LIN {X 0,Y 523.999,Z 356.213,A -85,B 0,C 180,E1 -4851.516,E2 -4851.516} C_VEL
LIN {X 0,Y 524.077,Z 356.199,A -85,B 0,C 180,E1 -4854.614,E2 -4854.614} C_VEL
LIN {X 0,Y 524.103,Z 356.198,A -85,B 0,C 180,E1 -4857.695,E2 -4857.695} C_VEL
LIN {X 0,Y 524.118,Z 356.196,A -85,B 0,C 180,E1 -4860.769,E2 -4860.769} C_VEL
LIN {X 0,Y 524.069,Z 356.203,A -85,B 0,C 180,E1 -4863.075,E2 -4863.075} C_VEL
LIN {X 0,Y 524.038,Z 356.203,A -85,B 0,C 180,E1 -4866.159,E2 -4866.159} C_VEL
LIN {X 0,Y 523.997,Z 356.217,A -85,B 0,C 180,E1 -4869.262,E2 -4869.262} C_VEL
LIN {X 0,Y 523.999,Z 356.208,A -85,B 0,C 180,E1 -4871.743,E2 -4871.743} C_VEL
LIN {X 0,Y 523.984,Z 356.219,A -85,B 0,C 180,E1 -4875.053,E2 -4875.053} C_VEL
LIN {X 0,Y 523.957,Z 356.214,A -85,B 0,C 180,E1 -4877.97,E2 -4877.97} C_VEL
LIN {X 0,Y 523.966,Z 356.212,A -85,B 0,C 180,E1 -4880.411,E2 -4880.411} C_VEL
LIN {X 0,Y 523.937,Z 356.224,A -85,B 0,C 180,E1 -4882.893,E2 -4882.893} C_VEL
LIN {X 0,Y 523.979,Z 356.211,A -85,B 0,C 180,E1 -4886.021,E2 -4886.021} C_VEL
LIN {X 0,Y 523.935,Z 356.225,A -85,B 0,C 180,E1 -4888.875,E2 -4888.875} C_VEL
LIN {X 0,Y 523.926,Z 356.22,A -85,B 0,C 180,E1 -4891.544,E2 -4891.544} C_VEL
LIN {X 0,Y 523.941,Z 356.214,A -85,B 0,C 180,E1 -4894.29,E2 -4894.29} C_VEL
LIN {X 0,Y 523.908,Z 356.225,A -85,B 0,C 180,E1 -4897.133,E2 -4897.133} C_VEL
LIN {X 0,Y 523.965,Z 356.214,A -85,B 0,C 180,E1 -4900.135,E2 -4900.135} C_VEL
LIN {X 0,Y 523.924,Z 356.223,A -85,B 0,C 180,E1 -4903.167,E2 -4903.167} C_VEL
LIN {X 0,Y 523.939,Z 356.217,A -85,B 0,C 180,E1 -4905.773,E2 -4905.773} C_VEL
LIN {X 0,Y 523.921,Z 356.223,A -85,B 0,C 180,E1 -4906.927,E2 -4906.927} C_VEL
LIN {X 0,Y 523.254,Z 356.304,A -85,B 0,C 180,E1 -4907.569,E2 -4907.569} C_VEL
LIN {X 0,Y 520.409,Z 356.664,A -85,B 0,C 180,E1 -4908.61,E2 -4908.61} C_VEL
LIN {X 0,Y 518.003,Z 356.963,A -85,B 0,C 180,E1 -4909.449,E2 -4909.449} C_VEL
LIN {X 0,Y 516.967,Z 357.09,A -85,B 0,C 180,E1 -4910.097,E2 -4910.097} C_VEL
LIN {X 0,Y 516.881,Z 357.101,A -85,B 0,C 180,E1 -4910.316,E2 -4910.316} C_VEL
LIN {X 0,Y 516.886,Z 357.102,A -85,B 0,C 180,E1 -4913.343,E2 -4913.343} C_VEL
LIN {X 0,Y 516.918,Z 357.18,A -85,B 0,C 180,E1 -4914.701,E2 -4914.701} C_VEL
LIN {X 0,Y 517.572,Z 361.395,A -85,B 0,C 180,E1 -4915.619,E2 -4915.619} C_VEL
LIN {X 0,Y 517.269,Z 376.326,A -85,B 0,C 180,E1 -4918.704,E2 -4918.704} C_VEL
LIN {X 0,Y 519.142,Z 386.126,A -85,B 0,C 180,E1 -4918.9,E2 -4918.9} C_VEL
LIN {X 0,Y 518.653,Z 482.307,A -85,B 0,C 180,E1 -4920.255,E2 -4920.255} C_VEL
LIN {X 0,Y 518.435,Z 495.531,A -85,B 0,C 180,E1 -4920.598,E2 -4920.598} C_VEL
LIN {X 0,Y 518.202,Z 508.654,A -85,B 0,C 180,E1 -4921.109,E2 -4921.109} C_VEL
LIN {X 0,Y 517.932,Z 520.368,A -85,B 0,C 180,E1 -4921.735,E2 -4921.735} C_VEL
LIN {X 0,Y 517.624,Z 531.628,A -85,B 0,C 180,E1 -4922.508,E2 -4922.508} C_VEL
LIN {X 0,Y 517.32,Z 541.648,A -85,B 0,C 180,E1 -4923.365,E2 -4923.365} C_VEL
LIN {X 0,Y 517.089,Z 549.864,A -85,B 0,C 180,E1 -4924.22,E2 -4924.22} C_VEL
LIN {X 0,Y 516.865,Z 558.043,A -85,B 0,C 180,E1 -4925.245,E2 -4925.245} C_VEL
LIN {X 0,Y 516.666,Z 565.201,A -85,B 0,C 180,E1 -4926.343,E2 -4926.343} C_VEL
LIN {X 0,Y 516.487,Z 572.285,A -85,B 0,C 180,E1 -4927.715,E2 -4927.715} C_VEL
LIN {X 0,Y 516.365,Z 576.909,A -85,B 0,C 180,E1 -4928.859,E2 -4928.859} C_VEL
LIN {X 0,Y 516.33,Z 580.762,A -85,B 0,C 180,E1 -4930.106,E2 -4930.106} C_VEL
LIN {X 0,Y 516.212,Z 582.707,A -85,B 0,C 180,E1 -4930.929,E2 -4930.929} C_VEL
LIN {X 0,Y 516.222,Z 584.92,A -85,B 0,C 180,E1 -4932.366,E2 -4932.366} C_VEL
LIN {X 0,Y 516.168,Z 585.709,A -85,B 0,C 180,E1 -4933.386,E2 -4933.386} C_VEL
LIN {X 0,Y 516.138,Z 585.826,A -85,B 0,C 180,E1 -4934.197,E2 -4934.197} C_VEL
LIN {X 0,Y 516.207,Z 585.427,A -85,B 0,C 180,E1 -4935.162,E2 -4935.162} C_VEL
LIN {X 0,Y 516.202,Z 583.697,A -85,B 0,C 180,E1 -4936.618,E2 -4936.618} C_VEL
LIN {X 0,Y 516.302,Z 581.187,A -85,B 0,C 180,E1 -4937.82,E2 -4937.82} C_VEL
LIN {X 0,Y 516.375,Z 577.665,A -85,B 0,C 180,E1 -4939.016,E2 -4939.016} C_VEL
LIN {X 0,Y 516.454,Z 573.038,A -85,B 0,C 180,E1 -4940.206,E2 -4940.206} C_VEL
LIN {X 0,Y 516.62,Z 566.055,A -85,B 0,C 180,E1 -4941.591,E2 -4941.591} C_VEL
LIN {X 0,Y 516.858,Z 558.51,A -85,B 0,C 180,E1 -4942.775,E2 -4942.775} C_VEL
LIN {X 0,Y 517.094,Z 549.072,A -85,B 0,C 180,E1 -4943.954,E2 -4943.954} C_VEL
LIN {X 0,Y 517.352,Z 539.351,A -85,B 0,C 180,E1 -4944.934,E2 -4944.934} C_VEL
LIN {X 0,Y 517.682,Z 528.486,A -85,B 0,C 180,E1 -4945.815,E2 -4945.815} C_VEL
LIN {X 0,Y 517.98,Z 517.863,A -85,B 0,C 180,E1 -4946.5,E2 -4946.5} C_VEL
LIN {X 0,Y 518.301,Z 505.089,A -85,B 0,C 180,E1 -4947.134,E2 -4947.134} C_VEL
LIN {X 0,Y 518.516,Z 492.947,A -85,B 0,C 180,E1 -4947.572,E2 -4947.572} C_VEL
LIN {X 0,Y 518.672,Z 480.556,A -85,B 0,C 180,E1 -4947.865,E2 -4947.865} C_VEL
LIN {X 0,Y 519.047,Z 385.536,A -85,B 0,C 180,E1 -4949.2,E2 -4949.2} C_VEL
LIN {X 0,Y 517.211,Z 376.145,A -85,B 0,C 180,E1 -4949.392,E2 -4949.392} C_VEL
LIN {X 0,Y 517.596,Z 361.894,A -85,B 0,C 180,E1 -4952.335,E2 -4952.335} C_VEL
LIN {X 0,Y 516.966,Z 357.094,A -85,B 0,C 180,E1 -4953.41,E2 -4953.41} C_VEL
LIN {X 0,Y 516.995,Z 357.083,A -85,B 0,C 180,E1 -4956.243,E2 -4956.243} C_VEL
LIN {X 0,Y 516.955,Z 357.095,A -85,B 0,C 180,E1 -4959.389,E2 -4959.389} C_VEL
LIN {X 0,Y 516.958,Z 357.088,A -85,B 0,C 180,E1 -4961.807,E2 -4961.807} C_VEL
LIN {X 0,Y 516.95,Z 357.092,A -85,B 0,C 180,E1 -4965.146,E2 -4965.146} C_VEL
LIN {X 0,Y 516.929,Z 357.089,A -85,B 0,C 180,E1 -4968.222,E2 -4968.222} C_VEL
LIN {X 0,Y 516.917,Z 357.092,A -85,B 0,C 180,E1 -4970.701,E2 -4970.701} C_VEL
LIN {X 0,Y 516.915,Z 357.091,A -85,B 0,C 180,E1 -4974.071,E2 -4974.071} C_VEL
LIN {X 0,Y 516.928,Z 357.091,A -85,B 0,C 180,E1 -4976.657,E2 -4976.657} C_VEL
LIN {X 0,Y 516.914,Z 357.095,A -85,B 0,C 180,E1 -4979.523,E2 -4979.523} C_VEL
LIN {X 0,Y 516.902,Z 357.093,A -85,B 0,C 180,E1 -4982.543,E2 -4982.543} C_VEL
LIN {X 0,Y 516.884,Z 357.101,A -85,B 0,C 180,E1 -4985.331,E2 -4985.331} C_VEL
LIN {X 0,Y 516.882,Z 357.095,A -85,B 0,C 180,E1 -4987.942,E2 -4987.942} C_VEL
LIN {X 0,Y 516.885,Z 357.098,A -85,B 0,C 180,E1 -4990.74,E2 -4990.74} C_VEL
LIN {X 0,Y 516.883,Z 357.1,A -85,B 0,C 180,E1 -4992.83,E2 -4992.83} C_VEL
LIN {X 0,Y 516.92,Z 357.099,A -85,B 0,C 180,E1 -4995.009,E2 -4995.009} C_VEL
LIN {X 0,Y 516.915,Z 357.092,A -85,B 0,C 180,E1 -4998.397,E2 -4998.397} C_VEL
LIN {X 0,Y 516.88,Z 357.099,A -85,B 0,C 180,E1 -5001.283,E2 -5001.283} C_VEL
LIN {X 0,Y 516.886,Z 357.095,A -85,B 0,C 180,E1 -5004.22,E2 -5004.22} C_VEL
LIN {X 0,Y 516.893,Z 357.1,A -85,B 0,C 180,E1 -5007.052,E2 -5007.052} C_VEL
LIN {X 0,Y 516.887,Z 357.094,A -85,B 0,C 180,E1 -5009.795,E2 -5009.795} C_VEL
LIN {X 0,Y 516.924,Z 357.093,A -85,B 0,C 180,E1 -5012.467,E2 -5012.467} C_VEL
LIN {X 0,Y 516.905,Z 357.097,A -85,B 0,C 180,E1 -5015.071,E2 -5015.071} C_VEL
LIN {X 0,Y 516.879,Z 357.1,A -85,B 0,C 180,E1 -5018.462,E2 -5018.462} C_VEL
LIN {X 0,Y 516.898,Z 357.098,A -85,B 0,C 180,E1 -5020.954,E2 -5020.954} C_VEL
LIN {X 0,Y 516.91,Z 357.092,A -85,B 0,C 180,E1 -5023.41,E2 -5023.41} C_VEL
LIN {X 0,Y 516.887,Z 357.094,A -85,B 0,C 180,E1 -5025.833,E2 -5025.833} C_VEL
LIN {X 0,Y 516.956,Z 357.089,A -85,B 0,C 180,E1 -5028.233,E2 -5028.233} C_VEL
LIN {X 0,Y 516.964,Z 357.085,A -85,B 0,C 180,E1 -5031.399,E2 -5031.399} C_VEL
LIN {X 0,Y 517.035,Z 357.084,A -85,B 0,C 180,E1 -5034.54,E2 -5034.54} C_VEL
LIN {X 0,Y 517.075,Z 357.071,A -85,B 0,C 180,E1 -5037.663,E2 -5037.663} C_VEL
LIN {X 0,Y 517.086,Z 357.074,A -85,B 0,C 180,E1 -5040.779,E2 -5040.779} C_VEL
LIN {X 0,Y 517.008,Z 357.08,A -85,B 0,C 180,E1 -5043.117,E2 -5043.117} C_VEL
LIN {X 0,Y 517.001,Z 357.086,A -85,B 0,C 180,E1 -5046.243,E2 -5046.243} C_VEL
LIN {X 0,Y 516.949,Z 357.086,A -85,B 0,C 180,E1 -5049.389,E2 -5049.389} C_VEL
LIN {X 0,Y 516.947,Z 357.088,A -85,B 0,C 180,E1 -5051.81,E2 -5051.81} C_VEL
LIN {X 0,Y 516.934,Z 357.089,A -85,B 0,C 180,E1 -5055.147,E2 -5055.147} C_VEL
LIN {X 0,Y 516.917,Z 357.098,A -85,B 0,C 180,E1 -5058.222,E2 -5058.222} C_VEL
LIN {X 0,Y 516.904,Z 357.095,A -85,B 0,C 180,E1 -5060.702,E2 -5060.702} C_VEL
LIN {X 0,Y 516.903,Z 357.098,A -85,B 0,C 180,E1 -5064.072,E2 -5064.072} C_VEL
LIN {X 0,Y 516.921,Z 357.093,A -85,B 0,C 180,E1 -5066.658,E2 -5066.658} C_VEL
LIN {X 0,Y 516.917,Z 357.091,A -85,B 0,C 180,E1 -5069.527,E2 -5069.527} C_VEL
LIN {X 0,Y 516.894,Z 357.097,A -85,B 0,C 180,E1 -5072.545,E2 -5072.545} C_VEL
LIN {X 0,Y 516.877,Z 357.096,A -85,B 0,C 180,E1 -5075.333,E2 -5075.333} C_VEL
LIN {X 0,Y 516.876,Z 357.102,A -85,B 0,C 180,E1 -5077.944,E2 -5077.944} C_VEL
LIN {X 0,Y 516.899,Z 357.094,A -85,B 0,C 180,E1 -5080.74,E2 -5080.74} C_VEL
LIN {X 0,Y 516.878,Z 357.102,A -85,B 0,C 180,E1 -5083.904,E2 -5083.904} C_VEL
LIN {X 0,Y 516.878,Z 357.103,A -85,B 0,C 180,E1 -5086.108,E2 -5086.108} C_VEL
LIN {X 0,Y 516.909,Z 357.092,A -85,B 0,C 180,E1 -5089.262,E2 -5089.262} C_VEL
LIN {X 0,Y 516.88,Z 357.102,A -85,B 0,C 180,E1 -5092.057,E2 -5092.057} C_VEL
LIN {X 0,Y 516.894,Z 357.094,A -85,B 0,C 180,E1 -5095.177,E2 -5095.177} C_VEL
LIN {X 0,Y 516.883,Z 357.102,A -85,B 0,C 180,E1 -5097.977,E2 -5097.977} C_VEL
LIN {X 0,Y 516.936,Z 357.091,A -85,B 0,C 180,E1 -5100.697,E2 -5100.697} C_VEL
LIN {X 0,Y 516.943,Z 357.097,A -85,B 0,C 180,E1 -5103.804,E2 -5103.804} C_VEL
LIN {X 0,Y 516.979,Z 357.292,A -85,B 0,C 180,E1 -5104.754,E2 -5104.754} C_VEL
LIN {X 0,Y 518.678,Z 366.12,A -85,B 0,C 180,E1 -5106.228,E2 -5106.228} C_VEL
LIN {X 0,Y 518.204,Z 383.61,A -85,B 0,C 180,E1 -5108.937,E2 -5108.937} C_VEL
LIN {X 0,Y 517.69,Z 403.523,A -85,B 0,C 180,E1 -5111.973,E2 -5111.973} C_VEL
LIN {X 0,Y 517.314,Z 421.232,A -85,B 0,C 180,E1 -5114.631,E2 -5114.631} C_VEL
LIN {X 0,Y 519.105,Z 433.679,A -85,B 0,C 180,E1 -5114.86,E2 -5114.86} C_VEL
LIN {X 0,Y 518.63,Z 529.582,A -85,B 0,C 180,E1 -5116.207,E2 -5116.207} C_VEL
LIN {X 0,Y 518.369,Z 542.929,A -85,B 0,C 180,E1 -5116.55,E2 -5116.55} C_VEL
LIN {X 0,Y 518.05,Z 556.268,A -85,B 0,C 180,E1 -5117.065,E2 -5117.065} C_VEL
LIN {X 0,Y 517.745,Z 568.697,A -85,B 0,C 180,E1 -5117.733,E2 -5117.733} C_VEL
LIN {X 0,Y 517.479,Z 580.404,A -85,B 0,C 180,E1 -5118.544,E2 -5118.544} C_VEL
LIN {X 0,Y 517.163,Z 590.635,A -85,B 0,C 180,E1 -5119.429,E2 -5119.429} C_VEL
LIN {X 0,Y 516.901,Z 599.843,A -85,B 0,C 180,E1 -5120.413,E2 -5120.413} C_VEL
LIN {X 0,Y 516.667,Z 608.817,A -85,B 0,C 180,E1 -5121.592,E2 -5121.592} C_VEL
LIN {X 0,Y 516.509,Z 616.042,A -85,B 0,C 180,E1 -5122.77,E2 -5122.77} C_VEL
LIN {X 0,Y 516.423,Z 622.625,A -85,B 0,C 180,E1 -5124.142,E2 -5124.142} C_VEL
LIN {X 0,Y 516.271,Z 626.976,A -85,B 0,C 180,E1 -5125.315,E2 -5125.315} C_VEL
LIN {X 0,Y 516.37,Z 629.286,A -85,B 0,C 180,E1 -5126.098,E2 -5126.098} C_VEL
LIN {X 0,Y 516.282,Z 631.152,A -85,B 0,C 180,E1 -5126.879,E2 -5126.879} C_VEL
LIN {X 0,Y 516.26,Z 632.552,A -85,B 0,C 180,E1 -5127.659,E2 -5127.659} C_VEL
LIN {X 0,Y 516.16,Z 634.157,A -85,B 0,C 180,E1 -5129.22,E2 -5129.22} C_VEL
LIN {X 0,Y 516.158,Z 634.374,A -85,B 0,C 180,E1 -5130,E2 -5130} C_VEL
LIN {X 0,Y 516.192,Z 633.547,A -85,B 0,C 180,E1 -5131.56,E2 -5131.56} C_VEL
LIN {X 0,Y 516.26,Z 632.55,A -85,B 0,C 180,E1 -5132.341,E2 -5132.341} C_VEL
LIN {X 0,Y 516.282,Z 631.147,A -85,B 0,C 180,E1 -5133.121,E2 -5133.121} C_VEL
LIN {X 0,Y 516.313,Z 628.198,A -85,B 0,C 180,E1 -5134.293,E2 -5134.293} C_VEL
LIN {X 0,Y 516.376,Z 624.207,A -85,B 0,C 180,E1 -5135.467,E2 -5135.467} C_VEL
LIN {X 0,Y 516.474,Z 618.311,A -85,B 0,C 180,E1 -5136.791,E2 -5136.791} C_VEL
LIN {X 0,Y 516.606,Z 611.362,A -85,B 0,C 180,E1 -5138.015,E2 -5138.015} C_VEL
LIN {X 0,Y 516.798,Z 603.043,A -85,B 0,C 180,E1 -5139.194,E2 -5139.194} C_VEL
LIN {X 0,Y 517.056,Z 594.52,A -85,B 0,C 180,E1 -5140.177,E2 -5140.177} C_VEL
LIN {X 0,Y 517.376,Z 583.992,A -85,B 0,C 180,E1 -5141.161,E2 -5141.161} C_VEL
LIN {X 0,Y 517.655,Z 572.776,A -85,B 0,C 180,E1 -5142.004,E2 -5142.004} C_VEL
LIN {X 0,Y 517.988,Z 562.168,A -85,B 0,C 180,E1 -5142.637,E2 -5142.637} C_VEL
LIN {X 0,Y 518.225,Z 550.45,A -85,B 0,C 180,E1 -5143.179,E2 -5143.179} C_VEL
LIN {X 0,Y 518.473,Z 537.871,A -85,B 0,C 180,E1 -5143.597,E2 -5143.597} C_VEL
LIN {X 0,Y 518.683,Z 525.111,A -85,B 0,C 180,E1 -5143.866,E2 -5143.866} C_VEL
LIN {X 0,Y 518.991,Z 432.34,A -85,B 0,C 180,E1 -5145.161,E2 -5145.161} C_VEL
LIN {X 0,Y 517.327,Z 421.045,A -85,B 0,C 180,E1 -5145.377,E2 -5145.377} C_VEL
LIN {X 0,Y 517.765,Z 399.611,A -85,B 0,C 180,E1 -5148.601,E2 -5148.601} C_VEL
LIN {X 0,Y 518.261,Z 380.763,A -85,B 0,C 180,E1 -5151.477,E2 -5151.477} C_VEL
LIN {X 0,Y 518.63,Z 365.975,A -85,B 0,C 180,E1 -5153.774,E2 -5153.774} C_VEL
LIN {X 0,Y 516.971,Z 357.09,A -85,B 0,C 180,E1 -5155.274,E2 -5155.274} C_VEL
LIN {X 0,Y 516.925,Z 357.098,A -85,B 0,C 180,E1 -5158.414,E2 -5158.414} C_VEL
LIN {X 0,Y 516.892,Z 357.095,A -85,B 0,C 180,E1 -5161.109,E2 -5161.109} C_VEL
LIN {X 0,Y 516.912,Z 357.098,A -85,B 0,C 180,E1 -5163.966,E2 -5163.966} C_VEL
LIN {X 0,Y 516.881,Z 357.098,A -85,B 0,C 180,E1 -5166.745,E2 -5166.745} C_VEL
LIN {X 0,Y 516.909,Z 357.096,A -85,B 0,C 180,E1 -5169.718,E2 -5169.718} C_VEL
LIN {X 0,Y 516.882,Z 357.095,A -85,B 0,C 180,E1 -5172.757,E2 -5172.757} C_VEL
LIN {X 0,Y 516.918,Z 357.091,A -85,B 0,C 180,E1 -5175.009,E2 -5175.009} C_VEL
LIN {X 0,Y 516.918,Z 357.093,A -85,B 0,C 180,E1 -5178.397,E2 -5178.397} C_VEL
LIN {X 0,Y 516.901,Z 357.094,A -85,B 0,C 180,E1 -5181.286,E2 -5181.286} C_VEL
LIN {X 0,Y 516.884,Z 357.098,A -85,B 0,C 180,E1 -5184.221,E2 -5184.221} C_VEL
LIN {X 0,Y 516.891,Z 357.093,A -85,B 0,C 180,E1 -5187.053,E2 -5187.053} C_VEL
LIN {X 0,Y 516.895,Z 357.099,A -85,B 0,C 180,E1 -5189.796,E2 -5189.796} C_VEL
LIN {X 0,Y 516.922,Z 357.09,A -85,B 0,C 180,E1 -5192.467,E2 -5192.467} C_VEL
LIN {X 0,Y 516.903,Z 357.093,A -85,B 0,C 180,E1 -5195.072,E2 -5195.072} C_VEL
LIN {X 0,Y 516.878,Z 357.093,A -85,B 0,C 180,E1 -5198.462,E2 -5198.462} C_VEL
LIN {X 0,Y 516.896,Z 357.095,A -85,B 0,C 180,E1 -5200.955,E2 -5200.955} C_VEL
LIN {X 0,Y 516.909,Z 357.095,A -85,B 0,C 180,E1 -5203.41,E2 -5203.41} C_VEL
LIN {X 0,Y 516.897,Z 357.097,A -85,B 0,C 180,E1 -5205.834,E2 -5205.834} C_VEL
LIN {X 0,Y 516.948,Z 357.088,A -85,B 0,C 180,E1 -5209.028,E2 -5209.028} C_VEL
LIN {X 0,Y 516.969,Z 357.081,A -85,B 0,C 180,E1 -5212.187,E2 -5212.187} C_VEL
LIN {X 0,Y 517.024,Z 357.077,A -85,B 0,C 180,E1 -5214.54,E2 -5214.54} C_VEL
LIN {X 0,Y 517.076,Z 357.074,A -85,B 0,C 180,E1 -5217.663,E2 -5217.663} C_VEL
LIN {X 0,Y 517.088,Z 357.072,A -85,B 0,C 180,E1 -5220.779,E2 -5220.779} C_VEL
LIN {X 0,Y 517.01,Z 357.082,A -85,B 0,C 180,E1 -5223.117,E2 -5223.117} C_VEL
LIN {X 0,Y 517.002,Z 357.079,A -85,B 0,C 180,E1 -5226.243,E2 -5226.243} C_VEL
LIN {X 0,Y 516.951,Z 357.093,A -85,B 0,C 180,E1 -5229.39,E2 -5229.39} C_VEL
LIN {X 0,Y 516.948,Z 357.085,A -85,B 0,C 180,E1 -5231.811,E2 -5231.811} C_VEL
LIN {X 0,Y 516.935,Z 357.095,A -85,B 0,C 180,E1 -5235.147,E2 -5235.147} C_VEL
LIN {X 0,Y 516.919,Z 357.091,A -85,B 0,C 180,E1 -5238.223,E2 -5238.223} C_VEL
LIN {X 0,Y 516.908,Z 357.094,A -85,B 0,C 180,E1 -5240.702,E2 -5240.702} C_VEL
LIN {X 0,Y 516.885,Z 357.099,A -85,B 0,C 180,E1 -5243.223,E2 -5243.223} C_VEL
LIN {X 0,Y 516.938,Z 357.089,A -85,B 0,C 180,E1 -5246.198,E2 -5246.198} C_VEL
LIN {X 0,Y 516.917,Z 357.094,A -85,B 0,C 180,E1 -5249.305,E2 -5249.305} C_VEL
LIN {X 0,Y 516.896,Z 357.098,A -85,B 0,C 180,E1 -5252.545,E2 -5252.545} C_VEL
LIN {X 0,Y 516.879,Z 357.098,A -85,B 0,C 180,E1 -5255.333,E2 -5255.333} C_VEL
LIN {X 0,Y 516.878,Z 357.096,A -85,B 0,C 180,E1 -5257.944,E2 -5257.944} C_VEL
LIN {X 0,Y 516.901,Z 357.101,A -85,B 0,C 180,E1 -5260.741,E2 -5260.741} C_VEL
LIN {X 0,Y 516.881,Z 357.097,A -85,B 0,C 180,E1 -5263.904,E2 -5263.904} C_VEL
LIN {X 0,Y 516.881,Z 357.098,A -85,B 0,C 180,E1 -5266.108,E2 -5266.108} C_VEL
LIN {X 0,Y 516.916,Z 357.096,A -85,B 0,C 180,E1 -5268.399,E2 -5268.399} C_VEL
LIN {X 0,Y 516.881,Z 357.101,A -85,B 0,C 180,E1 -5270.316,E2 -5270.316} C_VEL
LIN {X 0,Y 516.212,Z 357.187,A -85,B 0,C 180,E1 -5270.967,E2 -5270.967} C_VEL
LIN {X 0,Y 513.363,Z 357.541,A -85,B 0,C 180,E1 -5272.022,E2 -5272.022} C_VEL
LIN {X 0,Y 510.955,Z 357.844,A -85,B 0,C 180,E1 -5272.873,E2 -5272.873} C_VEL
LIN {X 0,Y 509.92,Z 357.97,A -85,B 0,C 180,E1 -5273.529,E2 -5273.529} C_VEL
LIN {X 0,Y 509.834,Z 357.98,A -85,B 0,C 180,E1 -5273.752,E2 -5273.752} C_VEL
LIN {X 0,Y 509.867,Z 358.085,A -85,B 0,C 180,E1 -5274.556,E2 -5274.556} C_VEL
LIN {X 0,Y 510.609,Z 363.173,A -85,B 0,C 180,E1 -5275.674,E2 -5275.674} C_VEL
LIN {X 0,Y 510.286,Z 376.497,A -85,B 0,C 180,E1 -5278.466,E2 -5278.466} C_VEL
LIN {X 0,Y 512.262,Z 386.394,A -85,B 0,C 180,E1 -5278.691,E2 -5278.691} C_VEL
LIN {X 0,Y 511.757,Z 483.293,A -85,B 0,C 180,E1 -5280.081,E2 -5280.081} C_VEL
LIN {X 0,Y 511.515,Z 497.109,A -85,B 0,C 180,E1 -5280.455,E2 -5280.455} C_VEL
LIN {X 0,Y 511.291,Z 509.634,A -85,B 0,C 180,E1 -5280.963,E2 -5280.963} C_VEL
LIN {X 0,Y 510.996,Z 521.095,A -85,B 0,C 180,E1 -5281.591,E2 -5281.591} C_VEL
LIN {X 0,Y 510.637,Z 533.044,A -85,B 0,C 180,E1 -5282.434,E2 -5282.434} C_VEL
LIN {X 0,Y 510.326,Z 542.927,A -85,B 0,C 180,E1 -5283.308,E2 -5283.308} C_VEL
LIN {X 0,Y 510.034,Z 551.834,A -85,B 0,C 180,E1 -5284.276,E2 -5284.276} C_VEL
LIN {X 0,Y 509.738,Z 560.967,A -85,B 0,C 180,E1 -5285.503,E2 -5285.503} C_VEL
LIN {X 0,Y 509.568,Z 567.782,A -85,B 0,C 180,E1 -5286.64,E2 -5286.64} C_VEL
LIN {X 0,Y 509.413,Z 573.613,A -85,B 0,C 180,E1 -5287.848,E2 -5287.848} C_VEL
LIN {X 0,Y 509.29,Z 577.911,A -85,B 0,C 180,E1 -5288.975,E2 -5288.975} C_VEL
LIN {X 0,Y 509.233,Z 581.59,A -85,B 0,C 180,E1 -5290.238,E2 -5290.238} C_VEL
LIN {X 0,Y 509.123,Z 584.135,A -85,B 0,C 180,E1 -5291.489,E2 -5291.489} C_VEL
LIN {X 0,Y 509.157,Z 585.233,A -85,B 0,C 180,E1 -5292.322,E2 -5292.322} C_VEL
LIN {X 0,Y 509.088,Z 585.908,A -85,B 0,C 180,E1 -5293.148,E2 -5293.148} C_VEL
LIN {X 0,Y 509.047,Z 586.175,A -85,B 0,C 180,E1 -5293.971,E2 -5293.971} C_VEL
LIN {X 0,Y 509.122,Z 585.816,A -85,B 0,C 180,E1 -5295.083,E2 -5295.083} C_VEL
LIN {X 0,Y 509.107,Z 584.373,A -85,B 0,C 180,E1 -5296.428,E2 -5296.428} C_VEL
LIN {X 0,Y 509.177,Z 582.943,A -85,B 0,C 180,E1 -5297.242,E2 -5297.242} C_VEL
LIN {X 0,Y 509.273,Z 579.919,A -85,B 0,C 180,E1 -5298.468,E2 -5298.468} C_VEL
LIN {X 0,Y 509.331,Z 575.914,A -85,B 0,C 180,E1 -5299.667,E2 -5299.667} C_VEL
LIN {X 0,Y 509.505,Z 569.695,A -85,B 0,C 180,E1 -5301.073,E2 -5301.073} C_VEL
LIN {X 0,Y 509.713,Z 562.938,A -85,B 0,C 180,E1 -5302.274,E2 -5302.274} C_VEL
LIN {X 0,Y 509.932,Z 554.842,A -85,B 0,C 180,E1 -5303.437,E2 -5303.437} C_VEL
LIN {X 0,Y 510.185,Z 545.962,A -85,B 0,C 180,E1 -5304.467,E2 -5304.467} C_VEL
LIN {X 0,Y 510.534,Z 535.379,A -85,B 0,C 180,E1 -5305.46,E2 -5305.46} C_VEL
LIN {X 0,Y 510.849,Z 524.879,A -85,B 0,C 180,E1 -5306.253,E2 -5306.253} C_VEL
LIN {X 0,Y 511.256,Z 513.128,A -85,B 0,C 180,E1 -5306.947,E2 -5306.947} C_VEL
LIN {X 0,Y 511.452,Z 501.053,A -85,B 0,C 180,E1 -5307.49,E2 -5307.49} C_VEL
LIN {X 0,Y 511.682,Z 487.742,A -85,B 0,C 180,E1 -5307.909,E2 -5307.909} C_VEL
LIN {X 0,Y 511.847,Z 472.57,A -85,B 0,C 180,E1 -5308.18,E2 -5308.18} C_VEL
LIN {X 0,Y 512.249,Z 386.404,A -85,B 0,C 180,E1 -5309.398,E2 -5309.398} C_VEL
LIN {X 0,Y 510.241,Z 376.477,A -85,B 0,C 180,E1 -5309.605,E2 -5309.605} C_VEL
LIN {X 0,Y 510.612,Z 363.229,A -85,B 0,C 180,E1 -5312.366,E2 -5312.366} C_VEL
LIN {X 0,Y 510.232,Z 359.582,A -85,B 0,C 180,E1 -5313.158,E2 -5313.158} C_VEL
LIN {X 0,Y 509.917,Z 357.972,A -85,B 0,C 180,E1 -5313.556,E2 -5313.556} C_VEL
LIN {X 0,Y 509.943,Z 357.962,A -85,B 0,C 180,E1 -5316.33,E2 -5316.33} C_VEL
LIN {X 0,Y 509.913,Z 357.966,A -85,B 0,C 180,E1 -5318.72,E2 -5318.72} C_VEL
LIN {X 0,Y 509.91,Z 357.965,A -85,B 0,C 180,E1 -5321.931,E2 -5321.931} C_VEL
LIN {X 0,Y 509.899,Z 357.972,A -85,B 0,C 180,E1 -5325.241,E2 -5325.241} C_VEL
LIN {X 0,Y 509.887,Z 357.967,A -85,B 0,C 180,E1 -5327.998,E2 -5327.998} C_VEL
LIN {X 0,Y 509.854,Z 357.975,A -85,B 0,C 180,E1 -5331.001,E2 -5331.001} C_VEL
LIN {X 0,Y 509.841,Z 357.976,A -85,B 0,C 180,E1 -5333.562,E2 -5333.562} C_VEL
LIN {X 0,Y 509.914,Z 357.963,A -85,B 0,C 180,E1 -5336.378,E2 -5336.378} C_VEL
LIN {X 0,Y 509.879,Z 357.971,A -85,B 0,C 180,E1 -5338.843,E2 -5338.843} C_VEL
LIN {X 0,Y 509.827,Z 357.977,A -85,B 0,C 180,E1 -5341.589,E2 -5341.589} C_VEL
LIN {X 0,Y 509.855,Z 357.971,A -85,B 0,C 180,E1 -5344.412,E2 -5344.412} C_VEL
LIN {X 0,Y 509.82,Z 357.98,A -85,B 0,C 180,E1 -5347.34,E2 -5347.34} C_VEL
LIN {X 0,Y 509.838,Z 357.973,A -85,B 0,C 180,E1 -5350.381,E2 -5350.381} C_VEL
LIN {X 0,Y 509.823,Z 357.983,A -85,B 0,C 180,E1 -5353.061,E2 -5353.061} C_VEL
LIN {X 0,Y 509.828,Z 357.974,A -85,B 0,C 180,E1 -5355.791,E2 -5355.791} C_VEL
LIN {X 0,Y 509.856,Z 357.973,A -85,B 0,C 180,E1 -5358.574,E2 -5358.574} C_VEL
LIN {X 0,Y 509.848,Z 357.971,A -85,B 0,C 180,E1 -5361.785,E2 -5361.785} C_VEL
LIN {X 0,Y 509.841,Z 357.976,A -85,B 0,C 180,E1 -5364.622,E2 -5364.622} C_VEL
LIN {X 0,Y 509.86,Z 357.971,A -85,B 0,C 180,E1 -5367.48,E2 -5367.48} C_VEL
LIN {X 0,Y 509.852,Z 357.972,A -85,B 0,C 180,E1 -5370.273,E2 -5370.273} C_VEL
LIN {X 0,Y 509.881,Z 357.974,A -85,B 0,C 180,E1 -5372.944,E2 -5372.944} C_VEL
LIN {X 0,Y 509.863,Z 357.969,A -85,B 0,C 180,E1 -5375.573,E2 -5375.573} C_VEL
LIN {X 0,Y 509.815,Z 357.976,A -85,B 0,C 180,E1 -5378.148,E2 -5378.148} C_VEL
LIN {X 0,Y 509.858,Z 357.978,A -85,B 0,C 180,E1 -5380.681,E2 -5380.681} C_VEL
LIN {X 0,Y 509.879,Z 357.97,A -85,B 0,C 180,E1 -5383.174,E2 -5383.174} C_VEL
LIN {X 0,Y 509.856,Z 357.97,A -85,B 0,C 180,E1 -5385.634,E2 -5385.634} C_VEL
LIN {X 0,Y 509.909,Z 357.969,A -85,B 0,C 180,E1 -5388.874,E2 -5388.874} C_VEL
LIN {X 0,Y 509.943,Z 357.961,A -85,B 0,C 180,E1 -5392.078,E2 -5392.078} C_VEL
LIN {X 0,Y 509.985,Z 357.961,A -85,B 0,C 180,E1 -5394.464,E2 -5394.464} C_VEL
LIN {X 0,Y 510.046,Z 357.946,A -85,B 0,C 180,E1 -5397.631,E2 -5397.631} C_VEL
LIN {X 0,Y 510.056,Z 357.95,A -85,B 0,C 180,E1 -5400.789,E2 -5400.789} C_VEL
LIN {X 0,Y 509.95,Z 357.959,A -85,B 0,C 180,E1 -5403.16,E2 -5403.16} C_VEL
LIN {X 0,Y 509.969,Z 357.963,A -85,B 0,C 180,E1 -5406.33,E2 -5406.33} C_VEL
LIN {X 0,Y 509.909,Z 357.968,A -85,B 0,C 180,E1 -5408.72,E2 -5408.72} C_VEL
LIN {X 0,Y 509.895,Z 357.968,A -85,B 0,C 180,E1 -5411.932,E2 -5411.932} C_VEL
LIN {X 0,Y 509.884,Z 357.967,A -85,B 0,C 180,E1 -5415.242,E2 -5415.242} C_VEL
LIN {X 0,Y 509.879,Z 357.971,A -85,B 0,C 180,E1 -5418.001,E2 -5418.001} C_VEL
LIN {X 0,Y 509.842,Z 357.972,A -85,B 0,C 180,E1 -5421.002,E2 -5421.002} C_VEL
LIN {X 0,Y 509.828,Z 357.974,A -85,B 0,C 180,E1 -5423.563,E2 -5423.563} C_VEL
LIN {X 0,Y 509.905,Z 357.971,A -85,B 0,C 180,E1 -5426.38,E2 -5426.38} C_VEL
LIN {X 0,Y 509.878,Z 357.968,A -85,B 0,C 180,E1 -5428.844,E2 -5428.844} C_VEL
LIN {X 0,Y 509.819,Z 357.976,A -85,B 0,C 180,E1 -5431.59,E2 -5431.59} C_VEL
LIN {X 0,Y 509.848,Z 357.976,A -85,B 0,C 180,E1 -5434.414,E2 -5434.414} C_VEL
LIN {X 0,Y 509.813,Z 357.976,A -85,B 0,C 180,E1 -5437.341,E2 -5437.341} C_VEL
LIN {X 0,Y 509.856,Z 357.974,A -85,B 0,C 180,E1 -5440.381,E2 -5440.381} C_VEL
LIN {X 0,Y 509.835,Z 357.973,A -85,B 0,C 180,E1 -5443.065,E2 -5443.065} C_VEL
LIN {X 0,Y 509.826,Z 357.979,A -85,B 0,C 180,E1 -5445.793,E2 -5445.793} C_VEL
LIN {X 0,Y 509.863,Z 357.971,A -85,B 0,C 180,E1 -5448.576,E2 -5448.576} C_VEL
LIN {X 0,Y 509.854,Z 357.977,A -85,B 0,C 180,E1 -5451.786,E2 -5451.786} C_VEL
LIN {X 0,Y 509.845,Z 357.972,A -85,B 0,C 180,E1 -5454.624,E2 -5454.624} C_VEL
LIN {X 0,Y 509.865,Z 357.972,A -85,B 0,C 180,E1 -5457.482,E2 -5457.482} C_VEL
LIN {X 0,Y 509.881,Z 357.973,A -85,B 0,C 180,E1 -5460.27,E2 -5460.27} C_VEL
LIN {X 0,Y 509.886,Z 357.972,A -85,B 0,C 180,E1 -5462.945,E2 -5462.945} C_VEL
LIN {X 0,Y 509.936,Z 357.997,A -85,B 0,C 180,E1 -5464.544,E2 -5464.544} C_VEL
LIN {X 0,Y 511.783,Z 368.525,A -85,B 0,C 180,E1 -5466.318,E2 -5466.318} C_VEL
LIN {X 0,Y 511.138,Z 387.871,A -85,B 0,C 180,E1 -5469.347,E2 -5469.347} C_VEL
LIN {X 0,Y 510.575,Z 408.838,A -85,B 0,C 180,E1 -5472.58,E2 -5472.58} C_VEL
LIN {X 0,Y 510.318,Z 420.982,A -85,B 0,C 180,E1 -5474.417,E2 -5474.417} C_VEL
LIN {X 0,Y 512.252,Z 435.53,A -85,B 0,C 180,E1 -5474.683,E2 -5474.683} C_VEL
LIN {X 0,Y 511.735,Z 529.208,A -85,B 0,C 180,E1 -5476.018,E2 -5476.018} C_VEL
LIN {X 0,Y 511.476,Z 542.571,A -85,B 0,C 180,E1 -5476.365,E2 -5476.365} C_VEL
LIN {X 0,Y 511.14,Z 555.919,A -85,B 0,C 180,E1 -5476.887,E2 -5476.887} C_VEL
LIN {X 0,Y 510.824,Z 567.663,A -85,B 0,C 180,E1 -5477.52,E2 -5477.52} C_VEL
LIN {X 0,Y 510.515,Z 578.763,A -85,B 0,C 180,E1 -5478.285,E2 -5478.285} C_VEL
LIN {X 0,Y 510.199,Z 589.245,A -85,B 0,C 180,E1 -5479.183,E2 -5479.183} C_VEL
LIN {X 0,Y 509.903,Z 597.816,A -85,B 0,C 180,E1 -5480.079,E2 -5480.079} C_VEL
LIN {X 0,Y 509.682,Z 605.729,A -85,B 0,C 180,E1 -5481.076,E2 -5481.076} C_VEL
LIN {X 0,Y 509.476,Z 613.459,A -85,B 0,C 180,E1 -5482.271,E2 -5482.271} C_VEL
LIN {X 0,Y 509.317,Z 619.72,A -85,B 0,C 180,E1 -5483.474,E2 -5483.474} C_VEL
LIN {X 0,Y 509.243,Z 625.327,A -85,B 0,C 180,E1 -5484.853,E2 -5484.853} C_VEL
LIN {X 0,Y 509.275,Z 628.953,A -85,B 0,C 180,E1 -5486.044,E2 -5486.044} C_VEL
LIN {X 0,Y 509.201,Z 630.82,A -85,B 0,C 180,E1 -5486.835,E2 -5486.835} C_VEL
LIN {X 0,Y 509.189,Z 632.221,A -85,B 0,C 180,E1 -5487.627,E2 -5487.627} C_VEL
LIN {X 0,Y 509.073,Z 633.825,A -85,B 0,C 180,E1 -5489.209,E2 -5489.209} C_VEL
LIN {X 0,Y 509.069,Z 634.041,A -85,B 0,C 180,E1 -5490,E2 -5490} C_VEL
LIN {X 0,Y 509.112,Z 633.213,A -85,B 0,C 180,E1 -5491.582,E2 -5491.582} C_VEL
LIN {X 0,Y 509.189,Z 632.215,A -85,B 0,C 180,E1 -5492.373,E2 -5492.373} C_VEL
LIN {X 0,Y 509.201,Z 630.811,A -85,B 0,C 180,E1 -5493.165,E2 -5493.165} C_VEL
LIN {X 0,Y 509.206,Z 627.859,A -85,B 0,C 180,E1 -5494.353,E2 -5494.353} C_VEL
LIN {X 0,Y 509.294,Z 623.866,A -85,B 0,C 180,E1 -5495.543,E2 -5495.543} C_VEL
LIN {X 0,Y 509.407,Z 617.828,A -85,B 0,C 180,E1 -5496.914,E2 -5496.914} C_VEL
LIN {X 0,Y 509.551,Z 611.016,A -85,B 0,C 180,E1 -5498.127,E2 -5498.127} C_VEL
LIN {X 0,Y 509.753,Z 602.694,A -85,B 0,C 180,E1 -5499.323,E2 -5499.323} C_VEL
LIN {X 0,Y 510.025,Z 594.168,A -85,B 0,C 180,E1 -5500.319,E2 -5500.319} C_VEL
LIN {X 0,Y 510.387,Z 583.637,A -85,B 0,C 180,E1 -5501.316,E2 -5501.316} C_VEL
LIN {X 0,Y 510.665,Z 572.417,A -85,B 0,C 180,E1 -5502.171,E2 -5502.171} C_VEL
LIN {X 0,Y 511.039,Z 561.805,A -85,B 0,C 180,E1 -5502.812,E2 -5502.812} C_VEL
LIN {X 0,Y 511.297,Z 550.078,A -85,B 0,C 180,E1 -5503.361,E2 -5503.361} C_VEL
LIN {X 0,Y 511.579,Z 536.572,A -85,B 0,C 180,E1 -5503.809,E2 -5503.809} C_VEL
LIN {X 0,Y 511.79,Z 523.149,A -85,B 0,C 180,E1 -5504.082,E2 -5504.082} C_VEL
LIN {X 0,Y 512.112,Z 432.847,A -85,B 0,C 180,E1 -5505.358,E2 -5505.358} C_VEL
LIN {X 0,Y 510.288,Z 420.625,A -85,B 0,C 180,E1 -5505.605,E2 -5505.605} C_VEL
LIN {X 0,Y 510.762,Z 400.629,A -85,B 0,C 180,E1 -5508.657,E2 -5508.657} C_VEL
LIN {X 0,Y 511.307,Z 381.828,A -85,B 0,C 180,E1 -5511.572,E2 -5511.572} C_VEL
LIN {X 0,Y 511.743,Z 368.402,A -85,B 0,C 180,E1 -5513.684,E2 -5513.684} C_VEL
LIN {X 0,Y 510.122,Z 358.973,A -85,B 0,C 180,E1 -5515.282,E2 -5515.282} C_VEL
LIN {X 0,Y 509.936,Z 357.968,A -85,B 0,C 180,E1 -5515.456,E2 -5515.456} C_VEL
LIN {X 0,Y 509.886,Z 357.971,A -85,B 0,C 180,E1 -5518.843,E2 -5518.843} C_VEL
LIN {X 0,Y 509.826,Z 357.977,A -85,B 0,C 180,E1 -5521.589,E2 -5521.589} C_VEL
LIN {X 0,Y 509.852,Z 357.976,A -85,B 0,C 180,E1 -5524.412,E2 -5524.412} C_VEL
LIN {X 0,Y 509.817,Z 357.978,A -85,B 0,C 180,E1 -5527.34,E2 -5527.34} C_VEL
LIN {X 0,Y 509.874,Z 357.972,A -85,B 0,C 180,E1 -5530.378,E2 -5530.378} C_VEL
LIN {X 0,Y 509.82,Z 357.974,A -85,B 0,C 180,E1 -5533.062,E2 -5533.062} C_VEL
LIN {X 0,Y 509.826,Z 357.981,A -85,B 0,C 180,E1 -5535.792,E2 -5535.792} C_VEL
LIN {X 0,Y 509.86,Z 357.971,A -85,B 0,C 180,E1 -5538.575,E2 -5538.575} C_VEL
LIN {X 0,Y 509.853,Z 357.977,A -85,B 0,C 180,E1 -5541.662,E2 -5541.662} C_VEL
LIN {X 0,Y 509.84,Z 357.973,A -85,B 0,C 180,E1 -5544.623,E2 -5544.623} C_VEL
LIN {X 0,Y 509.859,Z 357.973,A -85,B 0,C 180,E1 -5547.481,E2 -5547.481} C_VEL
LIN {X 0,Y 509.874,Z 357.969,A -85,B 0,C 180,E1 -5550.268,E2 -5550.268} C_VEL
LIN {X 0,Y 509.879,Z 357.968,A -85,B 0,C 180,E1 -5552.944,E2 -5552.944} C_VEL
LIN {X 0,Y 509.862,Z 357.976,A -85,B 0,C 180,E1 -5555.574,E2 -5555.574} C_VEL
LIN {X 0,Y 509.814,Z 357.975,A -85,B 0,C 180,E1 -5558.148,E2 -5558.148} C_VEL
LIN {X 0,Y 509.856,Z 357.971,A -85,B 0,C 180,E1 -5560.681,E2 -5560.681} C_VEL
LIN {X 0,Y 509.879,Z 357.968,A -85,B 0,C 180,E1 -5563.175,E2 -5563.175} C_VEL
LIN {X 0,Y 509.864,Z 357.976,A -85,B 0,C 180,E1 -5565.634,E2 -5565.634} C_VEL
LIN {X 0,Y 509.908,Z 357.964,A -85,B 0,C 180,E1 -5568.875,E2 -5568.875} C_VEL
LIN {X 0,Y 509.943,Z 357.957,A -85,B 0,C 180,E1 -5572.078,E2 -5572.078} C_VEL
LIN {X 0,Y 509.975,Z 357.955,A -85,B 0,C 180,E1 -5574.464,E2 -5574.464} C_VEL
LIN {X 0,Y 510.047,Z 357.95,A -85,B 0,C 180,E1 -5577.631,E2 -5577.631} C_VEL
LIN {X 0,Y 510.058,Z 357.948,A -85,B 0,C 180,E1 -5580.79,E2 -5580.79} C_VEL
LIN {X 0,Y 509.952,Z 357.962,A -85,B 0,C 180,E1 -5583.16,E2 -5583.16} C_VEL
LIN {X 0,Y 509.97,Z 357.955,A -85,B 0,C 180,E1 -5586.33,E2 -5586.33} C_VEL
LIN {X 0,Y 509.911,Z 357.964,A -85,B 0,C 180,E1 -5588.721,E2 -5588.721} C_VEL
LIN {X 0,Y 509.896,Z 357.963,A -85,B 0,C 180,E1 -5591.932,E2 -5591.932} C_VEL
LIN {X 0,Y 509.885,Z 357.972,A -85,B 0,C 180,E1 -5595.242,E2 -5595.242} C_VEL
LIN {X 0,Y 509.881,Z 357.968,A -85,B 0,C 180,E1 -5598.002,E2 -5598.002} C_VEL
LIN {X 0,Y 509.85,Z 357.977,A -85,B 0,C 180,E1 -5601.002,E2 -5601.002} C_VEL
LIN {X 0,Y 509.843,Z 357.972,A -85,B 0,C 180,E1 -5603.563,E2 -5603.563} C_VEL
LIN {X 0,Y 509.907,Z 357.966,A -85,B 0,C 180,E1 -5606.38,E2 -5606.38} C_VEL
LIN {X 0,Y 509.872,Z 357.976,A -85,B 0,C 180,E1 -5608.845,E2 -5608.845} C_VEL
LIN {X 0,Y 509.82,Z 357.977,A -85,B 0,C 180,E1 -5611.591,E2 -5611.591} C_VEL
LIN {X 0,Y 509.85,Z 357.97,A -85,B 0,C 180,E1 -5614.414,E2 -5614.414} C_VEL
LIN {X 0,Y 509.815,Z 357.978,A -85,B 0,C 180,E1 -5617.341,E2 -5617.341} C_VEL
LIN {X 0,Y 509.857,Z 357.974,A -85,B 0,C 180,E1 -5620.381,E2 -5620.381} C_VEL
LIN {X 0,Y 509.838,Z 357.979,A -85,B 0,C 180,E1 -5623.065,E2 -5623.065} C_VEL
LIN {X 0,Y 509.829,Z 357.975,A -85,B 0,C 180,E1 -5625.793,E2 -5625.793} C_VEL
LIN {X 0,Y 509.858,Z 357.978,A -85,B 0,C 180,E1 -5628.576,E2 -5628.576} C_VEL
LIN {X 0,Y 509.852,Z 357.976,A -85,B 0,C 180,E1 -5631.787,E2 -5631.787} C_VEL
LIN {X 0,Y 509.834,Z 357.98,A -85,B 0,C 180,E1 -5633.752,E2 -5633.752} C_VEL
LIN {X 0,Y 509.549,Z 358.387,A -85,B 0,C 180,E1 -5634.189,E2 -5634.189} C_VEL
LIN {X 0,Y 508.378,Z 360.147,A -85,B 0,C 180,E1 -5634.812,E2 -5634.812} C_VEL
LIN {X 0,Y 506.757,Z 362.716,A -85,B 0,C 180,E1 -5635.396,E2 -5635.396} C_VEL
LIN {X 0,Y 503.827,Z 368.763,A -85,B 0,C 180,E1 -5636.553,E2 -5636.553} C_VEL
LIN {X 0,Y 503.462,Z 370.709,A -85,B 0,C 180,E1 -5636.952,E2 -5636.952} C_VEL
LIN {X 0,Y 503.328,Z 376.94,A -85,B 0,C 180,E1 -5638.266,E2 -5638.266} C_VEL
LIN {X 0,Y 505.473,Z 388.512,A -85,B 0,C 180,E1 -5638.505,E2 -5638.505} C_VEL
LIN {X 0,Y 504.897,Z 483.205,A -85,B 0,C 180,E1 -5639.879,E2 -5639.879} C_VEL
LIN {X 0,Y 504.66,Z 496.285,A -85,B 0,C 180,E1 -5640.228,E2 -5640.228} C_VEL
LIN {X 0,Y 504.395,Z 509.441,A -85,B 0,C 180,E1 -5640.756,E2 -5640.756} C_VEL
LIN {X 0,Y 504.052,Z 521.965,A -85,B 0,C 180,E1 -5641.452,E2 -5641.452} C_VEL
LIN {X 0,Y 503.714,Z 533.068,A -85,B 0,C 180,E1 -5642.248,E2 -5642.248} C_VEL
LIN {X 0,Y 503.34,Z 543.863,A -85,B 0,C 180,E1 -5643.219,E2 -5643.219} C_VEL
LIN {X 0,Y 502.973,Z 553.718,A -85,B 0,C 180,E1 -5644.332,E2 -5644.332} C_VEL
LIN {X 0,Y 502.716,Z 561.454,A -85,B 0,C 180,E1 -5645.406,E2 -5645.406} C_VEL
LIN {X 0,Y 502.536,Z 567.984,A -85,B 0,C 180,E1 -5646.512,E2 -5646.512} C_VEL
LIN {X 0,Y 502.369,Z 574.145,A -85,B 0,C 180,E1 -5647.808,E2 -5647.808} C_VEL
LIN {X 0,Y 502.221,Z 578.858,A -85,B 0,C 180,E1 -5649.094,E2 -5649.094} C_VEL
LIN {X 0,Y 502.129,Z 582.351,A -85,B 0,C 180,E1 -5650.372,E2 -5650.372} C_VEL
LIN {X 0,Y 502.062,Z 584.054,A -85,B 0,C 180,E1 -5651.219,E2 -5651.219} C_VEL
LIN {X 0,Y 502.048,Z 585.434,A -85,B 0,C 180,E1 -5652.16,E2 -5652.16} C_VEL
LIN {X 0,Y 501.98,Z 586.463,A -85,B 0,C 180,E1 -5653.74,E2 -5653.74} C_VEL
LIN {X 0,Y 502.027,Z 586.203,A -85,B 0,C 180,E1 -5655.007,E2 -5655.007} C_VEL
LIN {X 0,Y 502.026,Z 585.022,A -85,B 0,C 180,E1 -5656.233,E2 -5656.233} C_VEL
LIN {X 0,Y 502.081,Z 583.697,A -85,B 0,C 180,E1 -5657.058,E2 -5657.058} C_VEL
LIN {X 0,Y 502.183,Z 580.547,A -85,B 0,C 180,E1 -5658.422,E2 -5658.422} C_VEL
LIN {X 0,Y 502.261,Z 577.047,A -85,B 0,C 180,E1 -5659.519,E2 -5659.519} C_VEL
LIN {X 0,Y 502.388,Z 572.076,A -85,B 0,C 180,E1 -5660.742,E2 -5660.742} C_VEL
LIN {X 0,Y 502.575,Z 565.835,A -85,B 0,C 180,E1 -5661.962,E2 -5661.962} C_VEL
LIN {X 0,Y 502.843,Z 558.057,A -85,B 0,C 180,E1 -5663.174,E2 -5663.174} C_VEL
LIN {X 0,Y 503.155,Z 548.333,A -85,B 0,C 180,E1 -5664.389,E2 -5664.389} C_VEL
LIN {X 0,Y 503.495,Z 539.37,A -85,B 0,C 180,E1 -5665.296,E2 -5665.296} C_VEL
LIN {X 0,Y 503.812,Z 528.324,A -85,B 0,C 180,E1 -5666.201,E2 -5666.201} C_VEL
LIN {X 0,Y 504.185,Z 517.485,A -85,B 0,C 180,E1 -5666.904,E2 -5666.904} C_VEL
LIN {X 0,Y 504.501,Z 505.551,A -85,B 0,C 180,E1 -5667.505,E2 -5667.505} C_VEL
LIN {X 0,Y 504.775,Z 493.279,A -85,B 0,C 180,E1 -5667.955,E2 -5667.955} C_VEL
LIN {X 0,Y 504.936,Z 480.673,A -85,B 0,C 180,E1 -5668.255,E2 -5668.255} C_VEL
LIN {X 0,Y 505.428,Z 387.338,A -85,B 0,C 180,E1 -5669.602,E2 -5669.602} C_VEL
LIN {X 0,Y 503.297,Z 376.647,A -85,B 0,C 180,E1 -5669.85,E2 -5669.85} C_VEL
LIN {X 0,Y 503.598,Z 362.71,A -85,B 0,C 180,E1 -5672.8,E2 -5672.8} C_VEL
LIN {X 0,Y 502.834,Z 358.854,A -85,B 0,C 180,E1 -5673.706,E2 -5673.706} C_VEL
LIN {X 0,Y 502.893,Z 358.84,A -85,B 0,C 180,E1 -5676.419,E2 -5676.419} C_VEL
LIN {X 0,Y 502.873,Z 358.844,A -85,B 0,C 180,E1 -5678.843,E2 -5678.843} C_VEL
LIN {X 0,Y 502.852,Z 358.843,A -85,B 0,C 180,E1 -5682.101,E2 -5682.101} C_VEL
LIN {X 0,Y 502.854,Z 358.851,A -85,B 0,C 180,E1 -5685.399,E2 -5685.399} C_VEL
LIN {X 0,Y 502.845,Z 358.844,A -85,B 0,C 180,E1 -5688.12,E2 -5688.12} C_VEL
LIN {X 0,Y 502.833,Z 358.845,A -85,B 0,C 180,E1 -5690.535,E2 -5690.535} C_VEL
LIN {X 0,Y 502.801,Z 358.854,A -85,B 0,C 180,E1 -5693.04,E2 -5693.04} C_VEL
LIN {X 0,Y 502.844,Z 358.846,A -85,B 0,C 180,E1 -5695.675,E2 -5695.675} C_VEL
LIN {X 0,Y 502.842,Z 358.844,A -85,B 0,C 180,E1 -5698.372,E2 -5698.372} C_VEL
LIN {X 0,Y 502.798,Z 358.853,A -85,B 0,C 180,E1 -5701.499,E2 -5701.499} C_VEL
LIN {X 0,Y 502.808,Z 358.849,A -85,B 0,C 180,E1 -5704.444,E2 -5704.444} C_VEL
LIN {X 0,Y 502.782,Z 358.859,A -85,B 0,C 180,E1 -5707.177,E2 -5707.177} C_VEL
LIN {X 0,Y 502.788,Z 358.85,A -85,B 0,C 180,E1 -5710.014,E2 -5710.014} C_VEL
LIN {X 0,Y 502.801,Z 358.849,A -85,B 0,C 180,E1 -5712.198,E2 -5712.198} C_VEL
LIN {X 0,Y 502.798,Z 358.852,A -85,B 0,C 180,E1 -5715.467,E2 -5715.467} C_VEL
LIN {X 0,Y 502.827,Z 358.846,A -85,B 0,C 180,E1 -5717.863,E2 -5717.863} C_VEL
LIN {X 0,Y 502.799,Z 358.857,A -85,B 0,C 180,E1 -5721.023,E2 -5721.023} C_VEL
LIN {X 0,Y 502.781,Z 358.852,A -85,B 0,C 180,E1 -5724.166,E2 -5724.166} C_VEL
LIN {X 0,Y 502.828,Z 358.853,A -85,B 0,C 180,E1 -5726.992,E2 -5726.992} C_VEL
LIN {X 0,Y 502.809,Z 358.848,A -85,B 0,C 180,E1 -5730.064,E2 -5730.064} C_VEL
LIN {X 0,Y 502.829,Z 358.85,A -85,B 0,C 180,E1 -5732.533,E2 -5732.533} C_VEL
LIN {X 0,Y 502.822,Z 358.849,A -85,B 0,C 180,E1 -5735.298,E2 -5735.298} C_VEL
LIN {X 0,Y 502.777,Z 358.852,A -85,B 0,C 180,E1 -5737.826,E2 -5737.826} C_VEL
LIN {X 0,Y 502.818,Z 358.851,A -85,B 0,C 180,E1 -5740.4,E2 -5740.4} C_VEL
LIN {X 0,Y 502.829,Z 358.851,A -85,B 0,C 180,E1 -5742.931,E2 -5742.931} C_VEL
LIN {X 0,Y 502.836,Z 358.845,A -85,B 0,C 180,E1 -5745.429,E2 -5745.429} C_VEL
LIN {X 0,Y 502.873,Z 358.848,A -85,B 0,C 180,E1 -5748.716,E2 -5748.716} C_VEL
LIN {X 0,Y 502.893,Z 358.838,A -85,B 0,C 180,E1 -5751.966,E2 -5751.966} C_VEL
LIN {X 0,Y 502.939,Z 358.838,A -85,B 0,C 180,E1 -5754.386,E2 -5754.386} C_VEL
LIN {X 0,Y 503.016,Z 358.822,A -85,B 0,C 180,E1 -5757.598,E2 -5757.598} C_VEL
LIN {X 0,Y 503.017,Z 358.824,A -85,B 0,C 180,E1 -5760,E2 -5760} C_VEL
LIN {X 0,Y 503.016,Z 358.83,A -85,B 0,C 180,E1 -5762.402,E2 -5762.402} C_VEL
LIN {X 0,Y 502.93,Z 358.833,A -85,B 0,C 180,E1 -5765.613,E2 -5765.613} C_VEL
LIN {X 0,Y 502.893,Z 358.841,A -85,B 0,C 180,E1 -5768.033,E2 -5768.033} C_VEL
LIN {X 0,Y 502.872,Z 358.84,A -85,B 0,C 180,E1 -5771.283,E2 -5771.283} C_VEL
LIN {X 0,Y 502.836,Z 358.85,A -85,B 0,C 180,E1 -5774.571,E2 -5774.571} C_VEL
LIN {X 0,Y 502.853,Z 358.845,A -85,B 0,C 180,E1 -5777.907,E2 -5777.907} C_VEL
LIN {X 0,Y 502.82,Z 358.852,A -85,B 0,C 180,E1 -5780.537,E2 -5780.537} C_VEL
LIN {X 0,Y 502.788,Z 358.851,A -85,B 0,C 180,E1 -5783.041,E2 -5783.041} C_VEL
LIN {X 0,Y 502.833,Z 358.847,A -85,B 0,C 180,E1 -5785.676,E2 -5785.676} C_VEL
LIN {X 0,Y 502.835,Z 358.851,A -85,B 0,C 180,E1 -5788.373,E2 -5788.373} C_VEL
LIN {X 0,Y 502.79,Z 358.851,A -85,B 0,C 180,E1 -5791.5,E2 -5791.5} C_VEL
LIN {X 0,Y 502.8,Z 358.853,A -85,B 0,C 180,E1 -5794.445,E2 -5794.445} C_VEL
LIN {X 0,Y 502.775,Z 358.852,A -85,B 0,C 180,E1 -5797.179,E2 -5797.179} C_VEL
LIN {X 0,Y 502.821,Z 358.854,A -85,B 0,C 180,E1 -5800.012,E2 -5800.012} C_VEL
LIN {X 0,Y 502.818,Z 358.853,A -85,B 0,C 180,E1 -5802.203,E2 -5802.203} C_VEL
LIN {X 0,Y 502.796,Z 358.851,A -85,B 0,C 180,E1 -5805.469,E2 -5805.469} C_VEL
LIN {X 0,Y 502.826,Z 358.846,A -85,B 0,C 180,E1 -5809.004,E2 -5809.004} C_VEL
LIN {X 0,Y 502.795,Z 358.857,A -85,B 0,C 180,E1 -5812.047,E2 -5812.047} C_VEL
LIN {X 0,Y 502.808,Z 358.848,A -85,B 0,C 180,E1 -5815.036,E2 -5815.036} C_VEL
LIN {X 0,Y 502.787,Z 358.859,A -85,B 0,C 180,E1 -5817.917,E2 -5817.917} C_VEL
LIN {X 0,Y 502.839,Z 358.848,A -85,B 0,C 180,E1 -5820.714,E2 -5820.714} C_VEL
LIN {X 0,Y 502.862,Z 358.85,A -85,B 0,C 180,E1 -5823.44,E2 -5823.44} C_VEL
LIN {X 0,Y 502.897,Z 359.018,A -85,B 0,C 180,E1 -5824.386,E2 -5824.386} C_VEL
LIN {X 0,Y 504.85,Z 369.563,A -85,B 0,C 180,E1 -5826.19,E2 -5826.19} C_VEL
LIN {X 0,Y 504.147,Z 389.347,A -85,B 0,C 180,E1 -5829.331,E2 -5829.331} C_VEL
LIN {X 0,Y 503.551,Z 409.863,A -85,B 0,C 180,E1 -5832.538,E2 -5832.538} C_VEL
LIN {X 0,Y 503.293,Z 420.522,A -85,B 0,C 180,E1 -5834.19,E2 -5834.19} C_VEL
LIN {X 0,Y 505.399,Z 435.206,A -85,B 0,C 180,E1 -5834.47,E2 -5834.47} C_VEL
LIN {X 0,Y 504.856,Z 528.832,A -85,B 0,C 180,E1 -5835.823,E2 -5835.823} C_VEL
LIN {X 0,Y 504.548,Z 542.211,A -85,B 0,C 180,E1 -5836.174,E2 -5836.174} C_VEL
LIN {X 0,Y 504.204,Z 555.567,A -85,B 0,C 180,E1 -5836.704,E2 -5836.704} C_VEL
LIN {X 0,Y 503.869,Z 566.621,A -85,B 0,C 180,E1 -5837.3,E2 -5837.3} C_VEL
LIN {X 0,Y 503.503,Z 578.418,A -85,B 0,C 180,E1 -5838.119,E2 -5838.119} C_VEL
LIN {X 0,Y 503.21,Z 588.905,A -85,B 0,C 180,E1 -5839.03,E2 -5839.03} C_VEL
LIN {X 0,Y 502.872,Z 597.478,A -85,B 0,C 180,E1 -5839.939,E2 -5839.939} C_VEL
LIN {X 0,Y 502.631,Z 605.392,A -85,B 0,C 180,E1 -5840.95,E2 -5840.95} C_VEL
LIN {X 0,Y 502.398,Z 613.123,A -85,B 0,C 180,E1 -5842.161,E2 -5842.161} C_VEL
LIN {X 0,Y 502.236,Z 619.84,A -85,B 0,C 180,E1 -5843.482,E2 -5843.482} C_VEL
LIN {X 0,Y 502.175,Z 624.994,A -85,B 0,C 180,E1 -5844.781,E2 -5844.781} C_VEL
LIN {X 0,Y 502.164,Z 628.619,A -85,B 0,C 180,E1 -5845.987,E2 -5845.987} C_VEL
LIN {X 0,Y 502.122,Z 630.488,A -85,B 0,C 180,E1 -5846.791,E2 -5846.791} C_VEL
LIN {X 0,Y 502.12,Z 631.89,A -85,B 0,C 180,E1 -5847.594,E2 -5847.594} C_VEL
LIN {X 0,Y 501.99,Z 633.492,A -85,B 0,C 180,E1 -5849.198,E2 -5849.198} C_VEL
LIN {X 0,Y 501.983,Z 633.707,A -85,B 0,C 180,E1 -5850,E2 -5850} C_VEL
LIN {X 0,Y 502.036,Z 632.879,A -85,B 0,C 180,E1 -5851.604,E2 -5851.604} C_VEL
LIN {X 0,Y 502.12,Z 631.88,A -85,B 0,C 180,E1 -5852.406,E2 -5852.406} C_VEL
LIN {X 0,Y 502.122,Z 630.475,A -85,B 0,C 180,E1 -5853.209,E2 -5853.209} C_VEL
LIN {X 0,Y 502.104,Z 627.519,A -85,B 0,C 180,E1 -5854.415,E2 -5854.415} C_VEL
LIN {X 0,Y 502.211,Z 623.526,A -85,B 0,C 180,E1 -5855.622,E2 -5855.622} C_VEL
LIN {X 0,Y 502.333,Z 617.484,A -85,B 0,C 180,E1 -5857.011,E2 -5857.011} C_VEL
LIN {X 0,Y 502.482,Z 610.67,A -85,B 0,C 180,E1 -5858.242,E2 -5858.242} C_VEL
LIN {X 0,Y 502.719,Z 602.346,A -85,B 0,C 180,E1 -5859.454,E2 -5859.454} C_VEL
LIN {X 0,Y 502.994,Z 593.815,A -85,B 0,C 180,E1 -5860.465,E2 -5860.465} C_VEL
LIN {X 0,Y 503.406,Z 583.282,A -85,B 0,C 180,E1 -5861.475,E2 -5861.475} C_VEL
LIN {X 0,Y 503.679,Z 572.056,A -85,B 0,C 180,E1 -5862.343,E2 -5862.343} C_VEL
LIN {X 0,Y 504.066,Z 561.439,A -85,B 0,C 180,E1 -5862.992,E2 -5862.992} C_VEL
LIN {X 0,Y 504.354,Z 549.702,A -85,B 0,C 180,E1 -5863.549,E2 -5863.549} C_VEL
LIN {X 0,Y 504.697,Z 536.188,A -85,B 0,C 180,E1 -5864.001,E2 -5864.001} C_VEL
LIN {X 0,Y 504.897,Z 522.729,A -85,B 0,C 180,E1 -5864.278,E2 -5864.278} C_VEL
LIN {X 0,Y 505.354,Z 434.166,A -85,B 0,C 180,E1 -5865.544,E2 -5865.544} C_VEL
LIN {X 0,Y 503.262,Z 420.284,A -85,B 0,C 180,E1 -5865.827,E2 -5865.827} C_VEL
LIN {X 0,Y 503.791,Z 400.326,A -85,B 0,C 180,E1 -5868.925,E2 -5868.925} C_VEL
LIN {X 0,Y 504.372,Z 381.549,A -85,B 0,C 180,E1 -5871.884,E2 -5871.884} C_VEL
LIN {X 0,Y 504.82,Z 369.505,A -85,B 0,C 180,E1 -5873.811,E2 -5873.811} C_VEL
LIN {X 0,Y 502.877,Z 358.847,A -85,B 0,C 180,E1 -5875.673,E2 -5875.673} C_VEL
LIN {X 0,Y 502.842,Z 358.853,A -85,B 0,C 180,E1 -5878.372,E2 -5878.372} C_VEL
LIN {X 0,Y 502.797,Z 358.853,A -85,B 0,C 180,E1 -5881.499,E2 -5881.499} C_VEL
LIN {X 0,Y 502.805,Z 358.853,A -85,B 0,C 180,E1 -5884.444,E2 -5884.444} C_VEL
LIN {X 0,Y 502.779,Z 358.854,A -85,B 0,C 180,E1 -5887.178,E2 -5887.178} C_VEL
LIN {X 0,Y 502.831,Z 358.854,A -85,B 0,C 180,E1 -5890.01,E2 -5890.01} C_VEL
LIN {X 0,Y 502.769,Z 358.853,A -85,B 0,C 180,E1 -5893.23,E2 -5893.23} C_VEL
LIN {X 0,Y 502.785,Z 358.857,A -85,B 0,C 180,E1 -5895.661,E2 -5895.661} C_VEL
LIN {X 0,Y 502.83,Z 358.852,A -85,B 0,C 180,E1 -5897.864,E2 -5897.864} C_VEL
LIN {X 0,Y 502.816,Z 358.847,A -85,B 0,C 180,E1 -5901.025,E2 -5901.025} C_VEL
LIN {X 0,Y 502.779,Z 358.856,A -85,B 0,C 180,E1 -5904.167,E2 -5904.167} C_VEL
LIN {X 0,Y 502.826,Z 358.845,A -85,B 0,C 180,E1 -5906.993,E2 -5906.993} C_VEL
LIN {X 0,Y 502.823,Z 358.849,A -85,B 0,C 180,E1 -5910.061,E2 -5910.061} C_VEL
LIN {X 0,Y 502.828,Z 358.846,A -85,B 0,C 180,E1 -5912.533,E2 -5912.533} C_VEL
LIN {X 0,Y 502.82,Z 358.849,A -85,B 0,C 180,E1 -5915.298,E2 -5915.298} C_VEL
LIN {X 0,Y 502.785,Z 358.854,A -85,B 0,C 180,E1 -5917.827,E2 -5917.827} C_VEL
LIN {X 0,Y 502.817,Z 358.848,A -85,B 0,C 180,E1 -5920.4,E2 -5920.4} C_VEL
LIN {X 0,Y 502.827,Z 358.844,A -85,B 0,C 180,E1 -5922.932,E2 -5922.932} C_VEL
LIN {X 0,Y 502.842,Z 358.852,A -85,B 0,C 180,E1 -5925.429,E2 -5925.429} C_VEL
LIN {X 0,Y 502.872,Z 358.839,A -85,B 0,C 180,E1 -5928.717,E2 -5928.717} C_VEL
LIN {X 0,Y 502.893,Z 358.836,A -85,B 0,C 180,E1 -5931.967,E2 -5931.967} C_VEL
LIN {X 0,Y 502.931,Z 358.833,A -85,B 0,C 180,E1 -5934.387,E2 -5934.387} C_VEL
LIN {X 0,Y 503.016,Z 358.826,A -85,B 0,C 180,E1 -5937.598,E2 -5937.598} C_VEL
LIN {X 0,Y 503.017,Z 358.824,A -85,B 0,C 180,E1 -5940,E2 -5940} C_VEL
LIN {X 0,Y 503.017,Z 358.819,A -85,B 0,C 180,E1 -5942.402,E2 -5942.402} C_VEL
LIN {X 0,Y 502.94,Z 358.835,A -85,B 0,C 180,E1 -5945.614,E2 -5945.614} C_VEL
LIN {X 0,Y 502.894,Z 358.836,A -85,B 0,C 180,E1 -5948.034,E2 -5948.034} C_VEL
LIN {X 0,Y 502.873,Z 358.844,A -85,B 0,C 180,E1 -5951.284,E2 -5951.284} C_VEL
LIN {X 0,Y 502.837,Z 358.847,A -85,B 0,C 180,E1 -5954.571,E2 -5954.571} C_VEL
LIN {X 0,Y 502.854,Z 358.843,A -85,B 0,C 180,E1 -5957.908,E2 -5957.908} C_VEL
LIN {X 0,Y 502.823,Z 358.847,A -85,B 0,C 180,E1 -5960.537,E2 -5960.537} C_VEL
LIN {X 0,Y 502.799,Z 358.856,A -85,B 0,C 180,E1 -5963.041,E2 -5963.041} C_VEL
LIN {X 0,Y 502.836,Z 358.846,A -85,B 0,C 180,E1 -5965.676,E2 -5965.676} C_VEL
LIN {X 0,Y 502.835,Z 358.847,A -85,B 0,C 180,E1 -5968.373,E2 -5968.373} C_VEL
LIN {X 0,Y 502.791,Z 358.853,A -85,B 0,C 180,E1 -5971.5,E2 -5971.5} C_VEL
LIN {X 0,Y 502.803,Z 358.848,A -85,B 0,C 180,E1 -5974.446,E2 -5974.446} C_VEL
LIN {X 0,Y 502.777,Z 358.856,A -85,B 0,C 180,E1 -5977.179,E2 -5977.179} C_VEL
LIN {X 0,Y 502.813,Z 358.848,A -85,B 0,C 180,E1 -5980.013,E2 -5980.013} C_VEL
LIN {X 0,Y 502.827,Z 358.847,A -85,B 0,C 180,E1 -5982.204,E2 -5982.204} C_VEL
LIN {X 0,Y 502.799,Z 358.851,A -85,B 0,C 180,E1 -5985.469,E2 -5985.469} C_VEL
LIN {X 0,Y 502.829,Z 358.847,A -85,B 0,C 180,E1 -5987.865,E2 -5987.865} C_VEL
LIN {X 0,Y 502.802,Z 358.857,A -85,B 0,C 180,E1 -5991.025,E2 -5991.025} C_VEL
LIN {X 0,Y 502.839,Z 358.921,A -85,B 0,C 180,E1 -5994.389,E2 -5994.389} C_VEL
LIN {X 0,Y 503.606,Z 363.539,A -85,B 0,C 180,E1 -5995.424,E2 -5995.424} C_VEL
LIN {X 0,Y 503.462,Z 370.709,A -85,B 0,C 180,E1 -5996.952,E2 -5996.952} C_VEL
LIN {X 0,Y 503.168,Z 372.963,A -85,B 0,C 180,E1 -5997.308,E2 -5997.308} C_VEL
LIN {X 0,Y 502.594,Z 375.82,A -85,B 0,C 180,E1 -5997.602,E2 -5997.602} C_VEL
LIN {X 0,Y 501.443,Z 380.824,A -85,B 0,C 180,E1 -5997.936,E2 -5997.936} C_VEL
LIN {X 0,Y 500.189,Z 386.447,A -85,B 0,C 180,E1 -5998.167,E2 -5998.167} C_VEL
LIN {X 0,Y 498.884,Z 394.424,A -85,B 0,C 180,E1 -5998.361,E2 -5998.361} C_VEL
LIN {X 0,Y 498.618,Z 398.508,A -85,B 0,C 180,E1 -5998.426,E2 -5998.426} C_VEL
LIN {X 0,Y 498.037,Z 483.341,A -85,B 0,C 180,E1 -5999.675,E2 -5999.675} C_VEL
LIN {X 0,Y 497.779,Z 496.741,A -85,B 0,C 180,E1 -6000.037,E2 -6000.037} C_VEL
LIN {X 0,Y 497.542,Z 509.27,A -85,B 0,C 180,E1 -6000.546,E2 -6000.546} C_VEL
LIN {X 0,Y 497.203,Z 521.282,A -85,B 0,C 180,E1 -6001.209,E2 -6001.209} C_VEL
LIN {X 0,Y 496.809,Z 533.097,A -85,B 0,C 180,E1 -6002.058,E2 -6002.058} C_VEL
LIN {X 0,Y 496.414,Z 543.027,A -85,B 0,C 180,E1 -6002.948,E2 -6002.948} C_VEL
LIN {X 0,Y 496.061,Z 552.107,A -85,B 0,C 180,E1 -6003.948,E2 -6003.948} C_VEL
LIN {X 0,Y 495.747,Z 560.823,A -85,B 0,C 180,E1 -6005.136,E2 -6005.136} C_VEL
LIN {X 0,Y 495.497,Z 568.185,A -85,B 0,C 180,E1 -6006.379,E2 -6006.379} C_VEL
LIN {X 0,Y 495.329,Z 573.429,A -85,B 0,C 180,E1 -6007.475,E2 -6007.475} C_VEL
LIN {X 0,Y 495.17,Z 578.416,A -85,B 0,C 180,E1 -6008.782,E2 -6008.782} C_VEL
LIN {X 0,Y 495.088,Z 582.14,A -85,B 0,C 180,E1 -6010.082,E2 -6010.082} C_VEL
LIN {X 0,Y 494.999,Z 583.97,A -85,B 0,C 180,E1 -6010.941,E2 -6010.941} C_VEL
LIN {X 0,Y 494.96,Z 585.68,A -85,B 0,C 180,E1 -6012.055,E2 -6012.055} C_VEL
LIN {X 0,Y 494.894,Z 586.752,A -85,B 0,C 180,E1 -6013.5,E2 -6013.5} C_VEL
LIN {X 0,Y 494.944,Z 586.592,A -85,B 0,C 180,E1 -6014.924,E2 -6014.924} C_VEL
LIN {X 0,Y 494.961,Z 585.666,A -85,B 0,C 180,E1 -6016.032,E2 -6016.032} C_VEL
LIN {X 0,Y 494.982,Z 584.439,A -85,B 0,C 180,E1 -6016.869,E2 -6016.869} C_VEL
LIN {X 0,Y 495.106,Z 581.179,A -85,B 0,C 180,E1 -6018.367,E2 -6018.367} C_VEL
LIN {X 0,Y 495.213,Z 576.735,A -85,B 0,C 180,E1 -6019.782,E2 -6019.782} C_VEL
LIN {X 0,Y 495.398,Z 570.57,A -85,B 0,C 180,E1 -6021.228,E2 -6021.228} C_VEL
LIN {X 0,Y 495.651,Z 563.857,A -85,B 0,C 180,E1 -6022.464,E2 -6022.464} C_VEL
LIN {X 0,Y 495.935,Z 555.554,A -85,B 0,C 180,E1 -6023.695,E2 -6023.695} C_VEL
LIN {X 0,Y 496.222,Z 547.022,A -85,B 0,C 180,E1 -6024.718,E2 -6024.718} C_VEL
LIN {X 0,Y 496.612,Z 536.519,A -85,B 0,C 180,E1 -6025.739,E2 -6025.739} C_VEL
LIN {X 0,Y 496.973,Z 526.119,A -85,B 0,C 180,E1 -6026.554,E2 -6026.554} C_VEL
LIN {X 0,Y 497.43,Z 514.587,A -85,B 0,C 180,E1 -6027.267,E2 -6027.267} C_VEL
LIN {X 0,Y 497.686,Z 502.735,A -85,B 0,C 180,E1 -6027.825,E2 -6027.825} C_VEL
LIN {X 0,Y 497.958,Z 489.848,A -85,B 0,C 180,E1 -6028.256,E2 -6028.256} C_VEL
LIN {X 0,Y 498.104,Z 477.77,A -85,B 0,C 180,E1 -6028.509,E2 -6028.509} C_VEL
LIN {X 0,Y 498.5,Z 387.615,A -85,B 0,C 180,E1 -6029.823,E2 -6029.823} C_VEL
LIN {X 0,Y 496.332,Z 376.958,A -85,B 0,C 180,E1 -6030.076,E2 -6030.076} C_VEL
LIN {X 0,Y 496.645,Z 364.03,A -85,B 0,C 180,E1 -6032.839,E2 -6032.839} C_VEL
LIN {X 0,Y 495.77,Z 359.733,A -85,B 0,C 180,E1 -6033.861,E2 -6033.861} C_VEL
LIN {X 0,Y 495.845,Z 359.718,A -85,B 0,C 180,E1 -6036.511,E2 -6036.511} C_VEL
LIN {X 0,Y 495.843,Z 359.721,A -85,B 0,C 180,E1 -6038.969,E2 -6038.969} C_VEL
LIN {X 0,Y 495.834,Z 359.718,A -85,B 0,C 180,E1 -6042.034,E2 -6042.034} C_VEL
LIN {X 0,Y 495.829,Z 359.725,A -85,B 0,C 180,E1 -6045.451,E2 -6045.451} C_VEL
LIN {X 0,Y 495.811,Z 359.72,A -85,B 0,C 180,E1 -6048.247,E2 -6048.247} C_VEL
LIN {X 0,Y 495.778,Z 359.726,A -85,B 0,C 180,E1 -6050.756,E2 -6050.756} C_VEL
LIN {X 0,Y 495.757,Z 359.733,A -85,B 0,C 180,E1 -6053.386,E2 -6053.386} C_VEL
LIN {X 0,Y 495.794,Z 359.722,A -85,B 0,C 180,E1 -6056.067,E2 -6056.067} C_VEL
LIN {X 0,Y 495.774,Z 359.728,A -85,B 0,C 180,E1 -6058.814,E2 -6058.814} C_VEL
LIN {X 0,Y 495.76,Z 359.728,A -85,B 0,C 180,E1 -6061.725,E2 -6061.725} C_VEL
LIN {X 0,Y 495.778,Z 359.727,A -85,B 0,C 180,E1 -6064.694,E2 -6064.694} C_VEL
LIN {X 0,Y 495.732,Z 359.732,A -85,B 0,C 180,E1 -6067.56,E2 -6067.56} C_VEL
LIN {X 0,Y 495.766,Z 359.729,A -85,B 0,C 180,E1 -6070.699,E2 -6070.699} C_VEL
LIN {X 0,Y 495.732,Z 359.729,A -85,B 0,C 180,E1 -6074,E2 -6074} C_VEL
LIN {X 0,Y 495.755,Z 359.734,A -85,B 0,C 180,E1 -6077.119,E2 -6077.119} C_VEL
LIN {X 0,Y 495.756,Z 359.726,A -85,B 0,C 180,E1 -6079.952,E2 -6079.952} C_VEL
LIN {X 0,Y 495.727,Z 359.733,A -85,B 0,C 180,E1 -6082.552,E2 -6082.552} C_VEL
LIN {X 0,Y 495.78,Z 359.725,A -85,B 0,C 180,E1 -6085.456,E2 -6085.456} C_VEL
LIN {X 0,Y 495.753,Z 359.729,A -85,B 0,C 180,E1 -6088.363,E2 -6088.363} C_VEL
LIN {X 0,Y 495.782,Z 359.724,A -85,B 0,C 180,E1 -6091.506,E2 -6091.506} C_VEL
LIN {X 0,Y 495.793,Z 359.722,A -85,B 0,C 180,E1 -6093.932,E2 -6093.932} C_VEL
LIN {X 0,Y 495.758,Z 359.73,A -85,B 0,C 180,E1 -6097.137,E2 -6097.137} C_VEL
LIN {X 0,Y 495.771,Z 359.726,A -85,B 0,C 180,E1 -6100.109,E2 -6100.109} C_VEL
LIN {X 0,Y 495.781,Z 359.732,A -85,B 0,C 180,E1 -6102.681,E2 -6102.681} C_VEL
LIN {X 0,Y 495.781,Z 359.725,A -85,B 0,C 180,E1 -6105.217,E2 -6105.217} C_VEL
LIN {X 0,Y 495.846,Z 359.723,A -85,B 0,C 180,E1 -6108.554,E2 -6108.554} C_VEL
LIN {X 0,Y 495.865,Z 359.713,A -85,B 0,C 180,E1 -6111.852,E2 -6111.852} C_VEL
LIN {X 0,Y 495.895,Z 359.714,A -85,B 0,C 180,E1 -6114.306,E2 -6114.306} C_VEL
LIN {X 0,Y 495.985,Z 359.698,A -85,B 0,C 180,E1 -6117.563,E2 -6117.563} C_VEL
LIN {X 0,Y 495.988,Z 359.7,A -85,B 0,C 180,E1 -6120,E2 -6120} C_VEL
LIN {X 0,Y 495.985,Z 359.706,A -85,B 0,C 180,E1 -6122.436,E2 -6122.436} C_VEL
LIN {X 0,Y 495.887,Z 359.711,A -85,B 0,C 180,E1 -6125.693,E2 -6125.693} C_VEL
LIN {X 0,Y 495.864,Z 359.718,A -85,B 0,C 180,E1 -6128.148,E2 -6128.148} C_VEL
LIN {X 0,Y 495.845,Z 359.715,A -85,B 0,C 180,E1 -6131.445,E2 -6131.445} C_VEL
LIN {X 0,Y 495.781,Z 359.726,A -85,B 0,C 180,E1 -6134.783,E2 -6134.783} C_VEL
LIN {X 0,Y 495.779,Z 359.724,A -85,B 0,C 180,E1 -6137.319,E2 -6137.319} C_VEL
LIN {X 0,Y 495.769,Z 359.728,A -85,B 0,C 180,E1 -6139.89,E2 -6139.89} C_VEL
LIN {X 0,Y 495.757,Z 359.728,A -85,B 0,C 180,E1 -6142.863,E2 -6142.863} C_VEL
LIN {X 0,Y 495.792,Z 359.728,A -85,B 0,C 180,E1 -6146.068,E2 -6146.068} C_VEL
LIN {X 0,Y 495.773,Z 359.726,A -85,B 0,C 180,E1 -6148.815,E2 -6148.815} C_VEL
LIN {X 0,Y 495.752,Z 359.73,A -85,B 0,C 180,E1 -6151.727,E2 -6151.727} C_VEL
LIN {X 0,Y 495.77,Z 359.726,A -85,B 0,C 180,E1 -6154.696,E2 -6154.696} C_VEL
LIN {X 0,Y 495.727,Z 359.732,A -85,B 0,C 180,E1 -6157.562,E2 -6157.562} C_VEL
LIN {X 0,Y 495.788,Z 359.731,A -85,B 0,C 180,E1 -6160.053,E2 -6160.053} C_VEL
LIN {X 0,Y 495.758,Z 359.726,A -85,B 0,C 180,E1 -6162.88,E2 -6162.88} C_VEL
LIN {X 0,Y 495.73,Z 359.739,A -85,B 0,C 180,E1 -6166,E2 -6166} C_VEL
LIN {X 0,Y 495.782,Z 359.724,A -85,B 0,C 180,E1 -6169.303,E2 -6169.303} C_VEL
LIN {X 0,Y 495.761,Z 359.728,A -85,B 0,C 180,E1 -6171.41,E2 -6171.41} C_VEL
LIN {X 0,Y 495.756,Z 359.728,A -85,B 0,C 180,E1 -6174.464,E2 -6174.464} C_VEL
LIN {X 0,Y 495.768,Z 359.727,A -85,B 0,C 180,E1 -6177.407,E2 -6177.407} C_VEL
LIN {X 0,Y 495.781,Z 359.731,A -85,B 0,C 180,E1 -6180.255,E2 -6180.255} C_VEL
LIN {X 0,Y 495.823,Z 359.726,A -85,B 0,C 180,E1 -6183.251,E2 -6183.251} C_VEL
LIN {X 0,Y 495.846,Z 359.825,A -85,B 0,C 180,E1 -6184.19,E2 -6184.19} C_VEL
LIN {X 0,Y 497.888,Z 370.706,A -85,B 0,C 180,E1 -6186.08,E2 -6186.08} C_VEL
LIN {X 0,Y 497.241,Z 388.109,A -85,B 0,C 180,E1 -6188.883,E2 -6188.883} C_VEL
LIN {X 0,Y 496.64,Z 408.195,A -85,B 0,C 180,E1 -6192.075,E2 -6192.075} C_VEL
LIN {X 0,Y 496.275,Z 420.218,A -85,B 0,C 180,E1 -6193.963,E2 -6193.963} C_VEL
LIN {X 0,Y 498.537,Z 436.172,A -85,B 0,C 180,E1 -6194.27,E2 -6194.27} C_VEL
LIN {X 0,Y 497.959,Z 529.609,A -85,B 0,C 180,E1 -6195.649,E2 -6195.649} C_VEL
LIN {X 0,Y 497.646,Z 542.614,A -85,B 0,C 180,E1 -6196.005,E2 -6196.005} C_VEL
LIN {X 0,Y 497.274,Z 555.214,A -85,B 0,C 180,E1 -6196.515,E2 -6196.515} C_VEL
LIN {X 0,Y 496.938,Z 566.278,A -85,B 0,C 180,E1 -6197.12,E2 -6197.12} C_VEL
LIN {X 0,Y 496.51,Z 578.074,A -85,B 0,C 180,E1 -6197.949,E2 -6197.949} C_VEL
LIN {X 0,Y 496.197,Z 588.564,A -85,B 0,C 180,E1 -6198.873,E2 -6198.873} C_VEL
LIN {X 0,Y 495.854,Z 597.139,A -85,B 0,C 180,E1 -6199.795,E2 -6199.795} C_VEL
LIN {X 0,Y 495.56,Z 605.054,A -85,B 0,C 180,E1 -6200.82,E2 -6200.82} C_VEL
LIN {X 0,Y 495.341,Z 612.788,A -85,B 0,C 180,E1 -6202.049,E2 -6202.049} C_VEL
LIN {X 0,Y 495.164,Z 619.916,A -85,B 0,C 180,E1 -6203.48,E2 -6203.48} C_VEL
LIN {X 0,Y 495.107,Z 624.661,A -85,B 0,C 180,E1 -6204.706,E2 -6204.706} C_VEL
LIN {X 0,Y 495.055,Z 628.286,A -85,B 0,C 180,E1 -6205.93,E2 -6205.93} C_VEL
LIN {X 0,Y 495.045,Z 630.156,A -85,B 0,C 180,E1 -6206.745,E2 -6206.745} C_VEL
LIN {X 0,Y 495.024,Z 631.557,A -85,B 0,C 180,E1 -6207.559,E2 -6207.559} C_VEL
LIN {X 0,Y 494.91,Z 633.16,A -85,B 0,C 180,E1 -6209.186,E2 -6209.186} C_VEL
LIN {X 0,Y 494.901,Z 633.375,A -85,B 0,C 180,E1 -6210,E2 -6210} C_VEL
LIN {X 0,Y 494.963,Z 632.545,A -85,B 0,C 180,E1 -6211.627,E2 -6211.627} C_VEL
LIN {X 0,Y 495.024,Z 631.544,A -85,B 0,C 180,E1 -6212.441,E2 -6212.441} C_VEL
LIN {X 0,Y 495.045,Z 630.139,A -85,B 0,C 180,E1 -6213.255,E2 -6213.255} C_VEL
LIN {X 0,Y 495.009,Z 627.18,A -85,B 0,C 180,E1 -6214.479,E2 -6214.479} C_VEL
LIN {X 0,Y 495.127,Z 623.185,A -85,B 0,C 180,E1 -6215.702,E2 -6215.702} C_VEL
LIN {X 0,Y 495.256,Z 617.038,A -85,B 0,C 180,E1 -6217.133,E2 -6217.133} C_VEL
LIN {X 0,Y 495.428,Z 610.323,A -85,B 0,C 180,E1 -6218.36,E2 -6218.36} C_VEL
LIN {X 0,Y 495.681,Z 601.996,A -85,B 0,C 180,E1 -6219.59,E2 -6219.59} C_VEL
LIN {X 0,Y 495.981,Z 593.462,A -85,B 0,C 180,E1 -6220.615,E2 -6220.615} C_VEL
LIN {X 0,Y 496.425,Z 582.926,A -85,B 0,C 180,E1 -6221.638,E2 -6221.638} C_VEL
LIN {X 0,Y 496.699,Z 572.016,A -85,B 0,C 180,E1 -6222.496,E2 -6222.496} C_VEL
LIN {X 0,Y 497.142,Z 561.075,A -85,B 0,C 180,E1 -6223.176,E2 -6223.176} C_VEL
LIN {X 0,Y 497.437,Z 549.328,A -85,B 0,C 180,E1 -6223.741,E2 -6223.741} C_VEL
LIN {X 0,Y 497.788,Z 535.802,A -85,B 0,C 180,E1 -6224.2,E2 -6224.2} C_VEL
LIN {X 0,Y 498.014,Z 522.308,A -85,B 0,C 180,E1 -6224.48,E2 -6224.48} C_VEL
LIN {X 0,Y 498.478,Z 434.77,A -85,B 0,C 180,E1 -6225.75,E2 -6225.75} C_VEL
LIN {X 0,Y 496.262,Z 420.022,A -85,B 0,C 180,E1 -6226.045,E2 -6226.045} C_VEL
LIN {X 0,Y 496.855,Z 400.025,A -85,B 0,C 180,E1 -6229.2,E2 -6229.2} C_VEL
LIN {X 0,Y 497.555,Z 379.977,A -85,B 0,C 180,E1 -6232.418,E2 -6232.418} C_VEL
LIN {X 0,Y 497.877,Z 370.632,A -85,B 0,C 180,E1 -6233.943,E2 -6233.943} C_VEL
LIN {X 0,Y 495.839,Z 359.723,A -85,B 0,C 180,E1 -6235.895,E2 -6235.895} C_VEL
LIN {X 0,Y 495.78,Z 359.728,A -85,B 0,C 180,E1 -6238.814,E2 -6238.814} C_VEL
LIN {X 0,Y 495.759,Z 359.731,A -85,B 0,C 180,E1 -6241.726,E2 -6241.726} C_VEL
LIN {X 0,Y 495.775,Z 359.727,A -85,B 0,C 180,E1 -6244.695,E2 -6244.695} C_VEL
LIN {X 0,Y 495.731,Z 359.734,A -85,B 0,C 180,E1 -6247.56,E2 -6247.56} C_VEL
LIN {X 0,Y 495.797,Z 359.731,A -85,B 0,C 180,E1 -6250.052,E2 -6250.052} C_VEL
LIN {X 0,Y 495.722,Z 359.73,A -85,B 0,C 180,E1 -6252.882,E2 -6252.882} C_VEL
LIN {X 0,Y 495.732,Z 359.738,A -85,B 0,C 180,E1 -6255.999,E2 -6255.999} C_VEL
LIN {X 0,Y 495.764,Z 359.727,A -85,B 0,C 180,E1 -6258.704,E2 -6258.704} C_VEL
LIN {X 0,Y 495.758,Z 359.729,A -85,B 0,C 180,E1 -6261.409,E2 -6261.409} C_VEL
LIN {X 0,Y 495.751,Z 359.729,A -85,B 0,C 180,E1 -6264.463,E2 -6264.463} C_VEL
LIN {X 0,Y 495.763,Z 359.728,A -85,B 0,C 180,E1 -6267.405,E2 -6267.405} C_VEL
LIN {X 0,Y 495.774,Z 359.725,A -85,B 0,C 180,E1 -6270.254,E2 -6270.254} C_VEL
LIN {X 0,Y 495.826,Z 359.721,A -85,B 0,C 180,E1 -6273.248,E2 -6273.248} C_VEL
LIN {X 0,Y 495.745,Z 359.736,A -85,B 0,C 180,E1 -6275.725,E2 -6275.725} C_VEL
LIN {X 0,Y 495.739,Z 359.727,A -85,B 0,C 180,E1 -6278.371,E2 -6278.371} C_VEL
LIN {X 0,Y 495.776,Z 359.726,A -85,B 0,C 180,E1 -6280.971,E2 -6280.971} C_VEL
LIN {X 0,Y 495.772,Z 359.729,A -85,B 0,C 180,E1 -6283.53,E2 -6283.53} C_VEL
LIN {X 0,Y 495.789,Z 359.724,A -85,B 0,C 180,E1 -6286.056,E2 -6286.056} C_VEL
LIN {X 0,Y 495.845,Z 359.714,A -85,B 0,C 180,E1 -6288.555,E2 -6288.555} C_VEL
LIN {X 0,Y 495.864,Z 359.712,A -85,B 0,C 180,E1 -6291.852,E2 -6291.852} C_VEL
LIN {X 0,Y 495.888,Z 359.71,A -85,B 0,C 180,E1 -6294.307,E2 -6294.307} C_VEL
LIN {X 0,Y 495.985,Z 359.701,A -85,B 0,C 180,E1 -6297.564,E2 -6297.564} C_VEL
LIN {X 0,Y 495.988,Z 359.699,A -85,B 0,C 180,E1 -6300,E2 -6300} C_VEL
LIN {X 0,Y 495.986,Z 359.695,A -85,B 0,C 180,E1 -6302.437,E2 -6302.437} C_VEL
LIN {X 0,Y 495.896,Z 359.711,A -85,B 0,C 180,E1 -6305.694,E2 -6305.694} C_VEL
LIN {X 0,Y 495.865,Z 359.712,A -85,B 0,C 180,E1 -6308.148,E2 -6308.148} C_VEL
LIN {X 0,Y 495.847,Z 359.717,A -85,B 0,C 180,E1 -6311.446,E2 -6311.446} C_VEL
LIN {X 0,Y 495.782,Z 359.728,A -85,B 0,C 180,E1 -6314.783,E2 -6314.783} C_VEL
LIN {X 0,Y 495.781,Z 359.73,A -85,B 0,C 180,E1 -6317.319,E2 -6317.319} C_VEL
LIN {X 0,Y 495.771,Z 359.723,A -85,B 0,C 180,E1 -6319.891,E2 -6319.891} C_VEL
LIN {X 0,Y 495.758,Z 359.734,A -85,B 0,C 180,E1 -6322.863,E2 -6322.863} C_VEL
LIN {X 0,Y 495.793,Z 359.723,A -85,B 0,C 180,E1 -6326.068,E2 -6326.068} C_VEL
LIN {X 0,Y 495.767,Z 359.732,A -85,B 0,C 180,E1 -6328.816,E2 -6328.816} C_VEL
LIN {X 0,Y 495.753,Z 359.729,A -85,B 0,C 180,E1 -6331.727,E2 -6331.727} C_VEL
LIN {X 0,Y 495.772,Z 359.725,A -85,B 0,C 180,E1 -6334.696,E2 -6334.696} C_VEL
LIN {X 0,Y 495.727,Z 359.731,A -85,B 0,C 180,E1 -6337.562,E2 -6337.562} C_VEL
LIN {X 0,Y 495.775,Z 359.732,A -85,B 0,C 180,E1 -6340.7,E2 -6340.7} C_VEL
LIN {X 0,Y 495.732,Z 359.732,A -85,B 0,C 180,E1 -6343.696,E2 -6343.696} C_VEL
LIN {X 0,Y 495.733,Z 359.734,A -85,B 0,C 180,E1 -6346.306,E2 -6346.306} C_VEL
LIN {X 0,Y 495.766,Z 359.73,A -85,B 0,C 180,E1 -6349.301,E2 -6349.301} C_VEL
LIN {X 0,Y 495.732,Z 359.739,A -85,B 0,C 180,E1 -6352.44,E2 -6352.44} C_VEL
LIN {X 0,Y 495.764,Z 359.763,A -85,B 0,C 180,E1 -6354.21,E2 -6354.21} C_VEL
LIN {X 0,Y 496.668,Z 365.581,A -85,B 0,C 180,E1 -6355.528,E2 -6355.528} C_VEL
LIN {X 0,Y 496.399,Z 377.213,A -85,B 0,C 180,E1 -6358.028,E2 -6358.028} C_VEL
LIN {X 0,Y 498.555,Z 387.954,A -85,B 0,C 180,E1 -6358.268,E2 -6358.268} C_VEL
LIN {X 0,Y 498.618,Z 398.508,A -85,B 0,C 180,E1 -6358.426,E2 -6358.426} C_VEL
LIN {X 0,Y 497.889,Z 404.351,A -85,B 0,C 180,E1 -6358.488,E2 -6358.488} C_VEL
LIN {X 0,Y 492.28,Z 423.358,A -85,B 0,C 180,E1 -6358.582,E2 -6358.582} C_VEL
LIN {X 0,Y 491.591,Z 429.2,A -85,B 0,C 180,E1 -6358.647,E2 -6358.647} C_VEL
LIN {X 0,Y 491.183,Z 484.274,A -85,B 0,C 180,E1 -6359.48,E2 -6359.48} C_VEL
LIN {X 0,Y 490.904,Z 497.733,A -85,B 0,C 180,E1 -6359.856,E2 -6359.856} C_VEL
LIN {X 0,Y 490.628,Z 510.349,A -85,B 0,C 180,E1 -6360.384,E2 -6360.384} C_VEL
LIN {X 0,Y 490.223,Z 522.756,A -85,B 0,C 180,E1 -6361.096,E2 -6361.096} C_VEL
LIN {X 0,Y 489.818,Z 534.557,A -85,B 0,C 180,E1 -6361.973,E2 -6361.973} C_VEL
LIN {X 0,Y 489.386,Z 544.686,A -85,B 0,C 180,E1 -6362.921,E2 -6362.921} C_VEL
LIN {X 0,Y 489.01,Z 554.014,A -85,B 0,C 180,E1 -6364.002,E2 -6364.002} C_VEL
LIN {X 0,Y 488.711,Z 562.064,A -85,B 0,C 180,E1 -6365.147,E2 -6365.147} C_VEL
LIN {X 0,Y 488.42,Z 569.556,A -85,B 0,C 180,E1 -6366.466,E2 -6366.466} C_VEL
LIN {X 0,Y 488.249,Z 574.613,A -85,B 0,C 180,E1 -6367.577,E2 -6367.577} C_VEL
LIN {X 0,Y 488.08,Z 579.383,A -85,B 0,C 180,E1 -6368.901,E2 -6368.901} C_VEL
LIN {X 0,Y 488.019,Z 581.855,A -85,B 0,C 180,E1 -6369.78,E2 -6369.78} C_VEL
LIN {X 0,Y 487.932,Z 583.85,A -85,B 0,C 180,E1 -6370.654,E2 -6370.654} C_VEL
LIN {X 0,Y 487.893,Z 585.898,A -85,B 0,C 180,E1 -6371.939,E2 -6371.939} C_VEL
LIN {X 0,Y 487.806,Z 586.992,A -85,B 0,C 180,E1 -6373.253,E2 -6373.253} C_VEL
LIN {X 0,Y 487.866,Z 586.983,A -85,B 0,C 180,E1 -6374.837,E2 -6374.837} C_VEL
LIN {X 0,Y 487.875,Z 586.236,A -85,B 0,C 180,E1 -6375.825,E2 -6375.825} C_VEL
LIN {X 0,Y 487.89,Z 585.168,A -85,B 0,C 180,E1 -6376.675,E2 -6376.675} C_VEL
LIN {X 0,Y 487.968,Z 583.628,A -85,B 0,C 180,E1 -6377.524,E2 -6377.524} C_VEL
LIN {X 0,Y 488.07,Z 580.521,A -85,B 0,C 180,E1 -6378.791,E2 -6378.791} C_VEL
LIN {X 0,Y 488.152,Z 576.357,A -85,B 0,C 180,E1 -6380.052,E2 -6380.052} C_VEL
LIN {X 0,Y 488.382,Z 569.999,A -85,B 0,C 180,E1 -6381.518,E2 -6381.518} C_VEL
LIN {X 0,Y 488.717,Z 562.456,A -85,B 0,C 180,E1 -6382.869,E2 -6382.869} C_VEL
LIN {X 0,Y 488.99,Z 554.433,A -85,B 0,C 180,E1 -6384.019,E2 -6384.019} C_VEL
LIN {X 0,Y 489.302,Z 545.604,A -85,B 0,C 180,E1 -6385.056,E2 -6385.056} C_VEL
LIN {X 0,Y 489.729,Z 535.886,A -85,B 0,C 180,E1 -6385.988,E2 -6385.988} C_VEL
LIN {X 0,Y 490.094,Z 525.258,A -85,B 0,C 180,E1 -6386.815,E2 -6386.815} C_VEL
LIN {X 0,Y 490.543,Z 513.309,A -85,B 0,C 180,E1 -6387.537,E2 -6387.537} C_VEL
LIN {X 0,Y 490.813,Z 500.957,A -85,B 0,C 180,E1 -6388.102,E2 -6388.102} C_VEL
LIN {X 0,Y 491.068,Z 487.993,A -85,B 0,C 180,E1 -6388.514,E2 -6388.514} C_VEL
LIN {X 0,Y 491.259,Z 472.38,A -85,B 0,C 180,E1 -6388.796,E2 -6388.796} C_VEL
LIN {X 0,Y 491.755,Z 389.036,A -85,B 0,C 180,E1 -6390.026,E2 -6390.026} C_VEL
LIN {X 0,Y 489.35,Z 377.373,A -85,B 0,C 180,E1 -6390.283,E2 -6390.283} C_VEL
LIN {X 0,Y 489.677,Z 365.336,A -85,B 0,C 180,E1 -6392.879,E2 -6392.879} C_VEL
LIN {X 0,Y 488.722,Z 360.61,A -85,B 0,C 180,E1 -6393.968,E2 -6393.968} C_VEL
LIN {X 0,Y 488.797,Z 360.597,A -85,B 0,C 180,E1 -6396.605,E2 -6396.605} C_VEL
LIN {X 0,Y 488.785,Z 360.601,A -85,B 0,C 180,E1 -6399.1,E2 -6399.1} C_VEL
LIN {X 0,Y 488.795,Z 360.594,A -85,B 0,C 180,E1 -6402.115,E2 -6402.115} C_VEL
LIN {X 0,Y 488.782,Z 360.601,A -85,B 0,C 180,E1 -6405.554,E2 -6405.554} C_VEL
LIN {X 0,Y 488.76,Z 360.598,A -85,B 0,C 180,E1 -6408.441,E2 -6408.441} C_VEL
LIN {X 0,Y 488.711,Z 360.609,A -85,B 0,C 180,E1 -6411.07,E2 -6411.07} C_VEL
LIN {X 0,Y 488.697,Z 360.608,A -85,B 0,C 180,E1 -6413.745,E2 -6413.745} C_VEL
LIN {X 0,Y 488.794,Z 360.598,A -85,B 0,C 180,E1 -6416.943,E2 -6416.943} C_VEL
LIN {X 0,Y 488.712,Z 360.604,A -85,B 0,C 180,E1 -6420.362,E2 -6420.362} C_VEL
LIN {X 0,Y 488.737,Z 360.605,A -85,B 0,C 180,E1 -6423.484,E2 -6423.484} C_VEL
LIN {X 0,Y 488.69,Z 360.607,A -85,B 0,C 180,E1 -6426.355,E2 -6426.355} C_VEL
LIN {X 0,Y 488.701,Z 360.612,A -85,B 0,C 180,E1 -6429.253,E2 -6429.253} C_VEL
LIN {X 0,Y 488.707,Z 360.606,A -85,B 0,C 180,E1 -6431.599,E2 -6431.599} C_VEL
LIN {X 0,Y 488.71,Z 360.61,A -85,B 0,C 180,E1 -6434.8,E2 -6434.8} C_VEL
LIN {X 0,Y 488.694,Z 360.609,A -85,B 0,C 180,E1 -6437.474,E2 -6437.474} C_VEL
LIN {X 0,Y 488.729,Z 360.603,A -85,B 0,C 180,E1 -6439.676,E2 -6439.676} C_VEL
LIN {X 0,Y 488.678,Z 360.615,A -85,B 0,C 180,E1 -6442.84,E2 -6442.84} C_VEL
LIN {X 0,Y 488.73,Z 360.602,A -85,B 0,C 180,E1 -6445.887,E2 -6445.887} C_VEL
LIN {X 0,Y 488.689,Z 360.615,A -85,B 0,C 180,E1 -6448.82,E2 -6448.82} C_VEL
LIN {X 0,Y 488.739,Z 360.601,A -85,B 0,C 180,E1 -6451.67,E2 -6451.67} C_VEL
LIN {X 0,Y 488.744,Z 360.604,A -85,B 0,C 180,E1 -6454.444,E2 -6454.444} C_VEL
LIN {X 0,Y 488.721,Z 360.606,A -85,B 0,C 180,E1 -6457.153,E2 -6457.153} C_VEL
LIN {X 0,Y 488.721,Z 360.603,A -85,B 0,C 180,E1 -6459.81,E2 -6459.81} C_VEL
LIN {X 0,Y 488.727,Z 360.606,A -85,B 0,C 180,E1 -6462.423,E2 -6462.423} C_VEL
LIN {X 0,Y 488.753,Z 360.603,A -85,B 0,C 180,E1 -6464.999,E2 -6464.999} C_VEL
LIN {X 0,Y 488.799,Z 360.598,A -85,B 0,C 180,E1 -6468.387,E2 -6468.387} C_VEL
LIN {X 0,Y 488.809,Z 360.592,A -85,B 0,C 180,E1 -6471.733,E2 -6471.733} C_VEL
LIN {X 0,Y 488.853,Z 360.59,A -85,B 0,C 180,E1 -6474.224,E2 -6474.224} C_VEL
LIN {X 0,Y 488.953,Z 360.574,A -85,B 0,C 180,E1 -6477.528,E2 -6477.528} C_VEL
LIN {X 0,Y 488.967,Z 360.576,A -85,B 0,C 180,E1 -6480.823,E2 -6480.823} C_VEL
LIN {X 0,Y 488.953,Z 360.583,A -85,B 0,C 180,E1 -6482.471,E2 -6482.471} C_VEL
LIN {X 0,Y 488.846,Z 360.588,A -85,B 0,C 180,E1 -6485.776,E2 -6485.776} C_VEL
LIN {X 0,Y 488.809,Z 360.598,A -85,B 0,C 180,E1 -6488.266,E2 -6488.266} C_VEL
LIN {X 0,Y 488.798,Z 360.594,A -85,B 0,C 180,E1 -6491.612,E2 -6491.612} C_VEL
LIN {X 0,Y 488.752,Z 360.6,A -85,B 0,C 180,E1 -6495.001,E2 -6495.001} C_VEL
LIN {X 0,Y 488.746,Z 360.607,A -85,B 0,C 180,E1 -6498.442,E2 -6498.442} C_VEL
LIN {X 0,Y 488.698,Z 360.606,A -85,B 0,C 180,E1 -6501.071,E2 -6501.071} C_VEL
LIN {X 0,Y 488.685,Z 360.609,A -85,B 0,C 180,E1 -6503.746,E2 -6503.746} C_VEL
LIN {X 0,Y 488.791,Z 360.595,A -85,B 0,C 180,E1 -6506.946,E2 -6506.946} C_VEL
LIN {X 0,Y 488.712,Z 360.61,A -85,B 0,C 180,E1 -6510.365,E2 -6510.365} C_VEL
LIN {X 0,Y 488.729,Z 360.603,A -85,B 0,C 180,E1 -6513.485,E2 -6513.485} C_VEL
LIN {X 0,Y 488.683,Z 360.613,A -85,B 0,C 180,E1 -6516.356,E2 -6516.356} C_VEL
LIN {X 0,Y 488.743,Z 360.6,A -85,B 0,C 180,E1 -6519.25,E2 -6519.25} C_VEL
LIN {X 0,Y 488.726,Z 360.605,A -85,B 0,C 180,E1 -6522.522,E2 -6522.522} C_VEL
LIN {X 0,Y 488.707,Z 360.605,A -85,B 0,C 180,E1 -6525.199,E2 -6525.199} C_VEL
LIN {X 0,Y 488.71,Z 360.607,A -85,B 0,C 180,E1 -6528.4,E2 -6528.4} C_VEL
LIN {X 0,Y 488.745,Z 360.6,A -85,B 0,C 180,E1 -6530.942,E2 -6530.942} C_VEL
LIN {X 0,Y 488.684,Z 360.615,A -85,B 0,C 180,E1 -6533.869,E2 -6533.869} C_VEL
LIN {X 0,Y 488.738,Z 360.601,A -85,B 0,C 180,E1 -6536.878,E2 -6536.878} C_VEL
LIN {X 0,Y 488.734,Z 360.609,A -85,B 0,C 180,E1 -6539.782,E2 -6539.782} C_VEL
LIN {X 0,Y 488.792,Z 360.601,A -85,B 0,C 180,E1 -6543.057,E2 -6543.057} C_VEL
LIN {X 0,Y 488.798,Z 360.625,A -85,B 0,C 180,E1 -6543.99,E2 -6543.99} C_VEL
LIN {X 0,Y 490.875,Z 371.555,A -85,B 0,C 180,E1 -6545.919,E2 -6545.919} C_VEL
LIN {X 0,Y 490.356,Z 387.415,A -85,B 0,C 180,E1 -6548.515,E2 -6548.515} C_VEL
LIN {X 0,Y 489.671,Z 407.856,A -85,B 0,C 180,E1 -6551.811,E2 -6551.811} C_VEL
LIN {X 0,Y 489.274,Z 420.106,A -85,B 0,C 180,E1 -6553.734,E2 -6553.734} C_VEL
LIN {X 0,Y 491.67,Z 437.063,A -85,B 0,C 180,E1 -6554.066,E2 -6554.066} C_VEL
LIN {X 0,Y 491.083,Z 529.15,A -85,B 0,C 180,E1 -6555.443,E2 -6555.443} C_VEL
LIN {X 0,Y 490.717,Z 542.969,A -85,B 0,C 180,E1 -6555.829,E2 -6555.829} C_VEL
LIN {X 0,Y 490.328,Z 555.881,A -85,B 0,C 180,E1 -6556.373,E2 -6556.373} C_VEL
LIN {X 0,Y 489.91,Z 567.667,A -85,B 0,C 180,E1 -6557.048,E2 -6557.048} C_VEL
LIN {X 0,Y 489.48,Z 579.028,A -85,B 0,C 180,E1 -6557.879,E2 -6557.879} C_VEL
LIN {X 0,Y 489.163,Z 589.277,A -85,B 0,C 180,E1 -6558.816,E2 -6558.816} C_VEL
LIN {X 0,Y 488.749,Z 598.489,A -85,B 0,C 180,E1 -6559.855,E2 -6559.855} C_VEL
LIN {X 0,Y 488.421,Z 607.469,A -85,B 0,C 180,E1 -6561.102,E2 -6561.102} C_VEL
LIN {X 0,Y 488.212,Z 614.701,A -85,B 0,C 180,E1 -6562.348,E2 -6562.348} C_VEL
LIN {X 0,Y 488.073,Z 620.074,A -85,B 0,C 180,E1 -6563.497,E2 -6563.497} C_VEL
LIN {X 0,Y 488.019,Z 624.328,A -85,B 0,C 180,E1 -6564.629,E2 -6564.629} C_VEL
LIN {X 0,Y 487.948,Z 627.952,A -85,B 0,C 180,E1 -6565.87,E2 -6565.87} C_VEL
LIN {X 0,Y 487.969,Z 629.824,A -85,B 0,C 180,E1 -6566.697,E2 -6566.697} C_VEL
LIN {X 0,Y 487.932,Z 631.224,A -85,B 0,C 180,E1 -6567.523,E2 -6567.523} C_VEL
LIN {X 0,Y 487.892,Z 632.222,A -85,B 0,C 180,E1 -6568.349,E2 -6568.349} C_VEL
LIN {X 0,Y 487.822,Z 633.042,A -85,B 0,C 180,E1 -6570,E2 -6570} C_VEL
LIN {X 0,Y 487.892,Z 632.211,A -85,B 0,C 180,E1 -6571.651,E2 -6571.651} C_VEL
LIN {X 0,Y 487.932,Z 631.208,A -85,B 0,C 180,E1 -6572.477,E2 -6572.477} C_VEL
LIN {X 0,Y 487.969,Z 629.802,A -85,B 0,C 180,E1 -6573.303,E2 -6573.303} C_VEL
LIN {X 0,Y 487.922,Z 626.842,A -85,B 0,C 180,E1 -6574.544,E2 -6574.544} C_VEL
LIN {X 0,Y 488.024,Z 622.843,A -85,B 0,C 180,E1 -6575.785,E2 -6575.785} C_VEL
LIN {X 0,Y 488.181,Z 616.694,A -85,B 0,C 180,E1 -6577.236,E2 -6577.236} C_VEL
LIN {X 0,Y 488.357,Z 609.976,A -85,B 0,C 180,E1 -6578.482,E2 -6578.482} C_VEL
LIN {X 0,Y 488.618,Z 601.645,A -85,B 0,C 180,E1 -6579.73,E2 -6579.73} C_VEL
LIN {X 0,Y 488.98,Z 593.11,A -85,B 0,C 180,E1 -6580.769,E2 -6580.769} C_VEL
LIN {X 0,Y 489.434,Z 582.578,A -85,B 0,C 180,E1 -6581.807,E2 -6581.807} C_VEL
LIN {X 0,Y 489.762,Z 571.02,A -85,B 0,C 180,E1 -6582.724,E2 -6582.724} C_VEL
LIN {X 0,Y 490.222,Z 558.811,A -85,B 0,C 180,E1 -6583.471,E2 -6583.471} C_VEL
LIN {X 0,Y 490.623,Z 546.425,A -85,B 0,C 180,E1 -6584.041,E2 -6584.041} C_VEL
LIN {X 0,Y 490.973,Z 533.707,A -85,B 0,C 180,E1 -6584.454,E2 -6584.454} C_VEL
LIN {X 0,Y 491.178,Z 520.369,A -85,B 0,C 180,E1 -6584.713,E2 -6584.713} C_VEL
LIN {X 0,Y 491.6,Z 435.328,A -85,B 0,C 180,E1 -6585.967,E2 -6585.967} C_VEL
LIN {X 0,Y 489.265,Z 419.663,A -85,B 0,C 180,E1 -6586.288,E2 -6586.288} C_VEL
LIN {X 0,Y 489.927,Z 399.762,A -85,B 0,C 180,E1 -6589.482,E2 -6589.482} C_VEL
LIN {X 0,Y 490.621,Z 381.088,A -85,B 0,C 180,E1 -6592.531,E2 -6592.531} C_VEL
LIN {X 0,Y 490.938,Z 371.768,A -85,B 0,C 180,E1 -6594.078,E2 -6594.078} C_VEL
LIN {X 0,Y 488.775,Z 360.604,A -85,B 0,C 180,E1 -6596.126,E2 -6596.126} C_VEL
LIN {X 0,Y 488.734,Z 360.606,A -85,B 0,C 180,E1 -6599.269,E2 -6599.269} C_VEL
LIN {X 0,Y 488.705,Z 360.614,A -85,B 0,C 180,E1 -6602.146,E2 -6602.146} C_VEL
LIN {X 0,Y 488.721,Z 360.604,A -85,B 0,C 180,E1 -6605.114,E2 -6605.114} C_VEL
LIN {X 0,Y 488.686,Z 360.611,A -85,B 0,C 180,E1 -6608.198,E2 -6608.198} C_VEL
LIN {X 0,Y 488.746,Z 360.605,A -85,B 0,C 180,E1 -6610.348,E2 -6610.348} C_VEL
LIN {X 0,Y 488.683,Z 360.612,A -85,B 0,C 180,E1 -6613.654,E2 -6613.654} C_VEL
LIN {X 0,Y 488.712,Z 360.608,A -85,B 0,C 180,E1 -6616.348,E2 -6616.348} C_VEL
LIN {X 0,Y 488.731,Z 360.609,A -85,B 0,C 180,E1 -6619.676,E2 -6619.676} C_VEL
LIN {X 0,Y 488.677,Z 360.611,A -85,B 0,C 180,E1 -6622.277,E2 -6622.277} C_VEL
LIN {X 0,Y 488.722,Z 360.604,A -85,B 0,C 180,E1 -6625.051,E2 -6625.051} C_VEL
LIN {X 0,Y 488.7,Z 360.61,A -85,B 0,C 180,E1 -6628.045,E2 -6628.045} C_VEL
LIN {X 0,Y 488.726,Z 360.601,A -85,B 0,C 180,E1 -6630.73,E2 -6630.73} C_VEL
LIN {X 0,Y 488.759,Z 360.604,A -85,B 0,C 180,E1 -6633.528,E2 -6633.528} C_VEL
LIN {X 0,Y 488.685,Z 360.609,A -85,B 0,C 180,E1 -6636.254,E2 -6636.254} C_VEL
LIN {X 0,Y 488.737,Z 360.601,A -85,B 0,C 180,E1 -6639.175,E2 -6639.175} C_VEL
LIN {X 0,Y 488.75,Z 360.604,A -85,B 0,C 180,E1 -6641.627,E2 -6641.627} C_VEL
LIN {X 0,Y 488.755,Z 360.601,A -85,B 0,C 180,E1 -6645,E2 -6645} C_VEL
LIN {X 0,Y 488.798,Z 360.592,A -85,B 0,C 180,E1 -6648.388,E2 -6648.388} C_VEL
LIN {X 0,Y 488.809,Z 360.592,A -85,B 0,C 180,E1 -6651.734,E2 -6651.734} C_VEL
LIN {X 0,Y 488.847,Z 360.588,A -85,B 0,C 180,E1 -6654.224,E2 -6654.224} C_VEL
LIN {X 0,Y 488.953,Z 360.577,A -85,B 0,C 180,E1 -6657.529,E2 -6657.529} C_VEL
LIN {X 0,Y 488.96,Z 360.575,A -85,B 0,C 180,E1 -6660,E2 -6660} C_VEL
LIN {X 0,Y 488.953,Z 360.571,A -85,B 0,C 180,E1 -6662.472,E2 -6662.472} C_VEL
LIN {X 0,Y 488.854,Z 360.588,A -85,B 0,C 180,E1 -6665.776,E2 -6665.776} C_VEL
LIN {X 0,Y 488.81,Z 360.59,A -85,B 0,C 180,E1 -6668.267,E2 -6668.267} C_VEL
LIN {X 0,Y 488.8,Z 360.593,A -85,B 0,C 180,E1 -6671.613,E2 -6671.613} C_VEL
LIN {X 0,Y 488.753,Z 360.607,A -85,B 0,C 180,E1 -6675.001,E2 -6675.001} C_VEL
LIN {X 0,Y 488.747,Z 360.602,A -85,B 0,C 180,E1 -6678.443,E2 -6678.443} C_VEL
LIN {X 0,Y 488.733,Z 360.607,A -85,B 0,C 180,E1 -6681.07,E2 -6681.07} C_VEL
LIN {X 0,Y 488.694,Z 360.605,A -85,B 0,C 180,E1 -6683.746,E2 -6683.746} C_VEL
LIN {X 0,Y 488.793,Z 360.6,A -85,B 0,C 180,E1 -6686.946,E2 -6686.946} C_VEL
LIN {X 0,Y 488.704,Z 360.607,A -85,B 0,C 180,E1 -6690.364,E2 -6690.364} C_VEL
LIN {X 0,Y 488.731,Z 360.599,A -85,B 0,C 180,E1 -6693.485,E2 -6693.485} C_VEL
LIN {X 0,Y 488.685,Z 360.611,A -85,B 0,C 180,E1 -6696.357,E2 -6696.357} C_VEL
LIN {X 0,Y 488.734,Z 360.605,A -85,B 0,C 180,E1 -6699.252,E2 -6699.252} C_VEL
LIN {X 0,Y 488.733,Z 360.604,A -85,B 0,C 180,E1 -6702.522,E2 -6702.522} C_VEL
LIN {X 0,Y 488.7,Z 360.608,A -85,B 0,C 180,E1 -6705.977,E2 -6705.977} C_VEL
LIN {X 0,Y 488.718,Z 360.612,A -85,B 0,C 180,E1 -6708.587,E2 -6708.587} C_VEL
LIN {X 0,Y 488.681,Z 360.615,A -85,B 0,C 180,E1 -6711.801,E2 -6711.801} C_VEL
LIN {X 0,Y 488.778,Z 360.803,A -85,B 0,C 180,E1 -6714.069,E2 -6714.069} C_VEL
LIN {X 0,Y 489.729,Z 366.884,A -85,B 0,C 180,E1 -6715.47,E2 -6715.47} C_VEL
LIN {X 0,Y 489.405,Z 377.507,A -85,B 0,C 180,E1 -6717.779,E2 -6717.779} C_VEL
LIN {X 0,Y 491.827,Z 389.64,A -85,B 0,C 180,E1 -6718.063,E2 -6718.063} C_VEL
LIN {X 0,Y 491.591,Z 429.2,A -85,B 0,C 180,E1 -6718.647,E2 -6718.647} C_VEL
LIN {X 0,Y 490.909,Z 435.04,A -85,B 0,C 180,E1 -6718.711,E2 -6718.711} C_VEL
LIN {X 0,Y 485.332,Z 454.049,A -85,B 0,C 180,E1 -6718.81,E2 -6718.81} C_VEL
LIN {X 0,Y 484.589,Z 459.892,A -85,B 0,C 180,E1 -6718.873,E2 -6718.873} C_VEL
LIN {X 0,Y 484.329,Z 485.744,A -85,B 0,C 180,E1 -6719.291,E2 -6719.291} C_VEL
LIN {X 0,Y 484.07,Z 498.739,A -85,B 0,C 180,E1 -6719.671,E2 -6719.671} C_VEL
LIN {X 0,Y 483.716,Z 511.379,A -85,B 0,C 180,E1 -6720.218,E2 -6720.218} C_VEL
LIN {X 0,Y 483.288,Z 524.088,A -85,B 0,C 180,E1 -6720.971,E2 -6720.971} C_VEL
LIN {X 0,Y 482.905,Z 534.632,A -85,B 0,C 180,E1 -6721.772,E2 -6721.772} C_VEL
LIN {X 0,Y 482.463,Z 544.478,A -85,B 0,C 180,E1 -6722.697,E2 -6722.697} C_VEL
LIN {X 0,Y 482.032,Z 554.186,A -85,B 0,C 180,E1 -6723.83,E2 -6723.83} C_VEL
LIN {X 0,Y 481.712,Z 562.133,A -85,B 0,C 180,E1 -6724.97,E2 -6724.97} C_VEL
LIN {X 0,Y 481.397,Z 569.79,A -85,B 0,C 180,E1 -6726.33,E2 -6726.33} C_VEL
LIN {X 0,Y 481.166,Z 575.735,A -85,B 0,C 180,E1 -6727.682,E2 -6727.682} C_VEL
LIN {X 0,Y 481.005,Z 580.96,A -85,B 0,C 180,E1 -6729.247,E2 -6729.247} C_VEL
LIN {X 0,Y 480.865,Z 583.675,A -85,B 0,C 180,E1 -6730.358,E2 -6730.358} C_VEL
LIN {X 0,Y 480.799,Z 586.135,A -85,B 0,C 180,E1 -6731.83,E2 -6731.83} C_VEL
LIN {X 0,Y 480.72,Z 587.192,A -85,B 0,C 180,E1 -6732.999,E2 -6732.999} C_VEL
LIN {X 0,Y 480.703,Z 587.491,A -85,B 0,C 180,E1 -6733.872,E2 -6733.872} C_VEL
LIN {X 0,Y 480.763,Z 587.365,A -85,B 0,C 180,E1 -6734.758,E2 -6734.758} C_VEL
LIN {X 0,Y 480.801,Z 586.793,A -85,B 0,C 180,E1 -6735.612,E2 -6735.612} C_VEL
LIN {X 0,Y 480.788,Z 585.818,A -85,B 0,C 180,E1 -6736.475,E2 -6736.475} C_VEL
LIN {X 0,Y 480.855,Z 584.435,A -85,B 0,C 180,E1 -6737.336,E2 -6737.336} C_VEL
LIN {X 0,Y 480.993,Z 581.417,A -85,B 0,C 180,E1 -6738.658,E2 -6738.658} C_VEL
LIN {X 0,Y 481.073,Z 577.541,A -85,B 0,C 180,E1 -6739.904,E2 -6739.904} C_VEL
LIN {X 0,Y 481.319,Z 571.422,A -85,B 0,C 180,E1 -6741.393,E2 -6741.393} C_VEL
LIN {X 0,Y 481.593,Z 564.819,A -85,B 0,C 180,E1 -6742.652,E2 -6742.652} C_VEL
LIN {X 0,Y 481.922,Z 556.494,A -85,B 0,C 180,E1 -6743.931,E2 -6743.931} C_VEL
LIN {X 0,Y 482.25,Z 548.03,A -85,B 0,C 180,E1 -6744.984,E2 -6744.984} C_VEL
LIN {X 0,Y 482.689,Z 537.589,A -85,B 0,C 180,E1 -6746.034,E2 -6746.034} C_VEL
LIN {X 0,Y 483.101,Z 527.261,A -85,B 0,C 180,E1 -6746.873,E2 -6746.873} C_VEL
LIN {X 0,Y 483.607,Z 515.883,A -85,B 0,C 180,E1 -6747.605,E2 -6747.605} C_VEL
LIN {X 0,Y 483.885,Z 504.257,A -85,B 0,C 180,E1 -6748.179,E2 -6748.179} C_VEL
LIN {X 0,Y 484.184,Z 491.713,A -85,B 0,C 180,E1 -6748.622,E2 -6748.622} C_VEL
LIN {X 0,Y 484.39,Z 478.882,A -85,B 0,C 180,E1 -6748.909,E2 -6748.909} C_VEL
LIN {X 0,Y 484.941,Z 390.093,A -85,B 0,C 180,E1 -6750.238,E2 -6750.238} C_VEL
LIN {X 0,Y 482.389,Z 377.624,A -85,B 0,C 180,E1 -6750.526,E2 -6750.526} C_VEL
LIN {X 0,Y 482.724,Z 366.639,A -85,B 0,C 180,E1 -6752.921,E2 -6752.921} C_VEL
LIN {X 0,Y 481.678,Z 361.487,A -85,B 0,C 180,E1 -6754.131,E2 -6754.131} C_VEL
LIN {X 0,Y 481.754,Z 361.475,A -85,B 0,C 180,E1 -6756.702,E2 -6756.702} C_VEL
LIN {X 0,Y 481.742,Z 361.48,A -85,B 0,C 180,E1 -6759.234,E2 -6759.234} C_VEL
LIN {X 0,Y 481.759,Z 361.47,A -85,B 0,C 180,E1 -6762.199,E2 -6762.199} C_VEL
LIN {X 0,Y 481.73,Z 361.478,A -85,B 0,C 180,E1 -6765.658,E2 -6765.658} C_VEL
LIN {X 0,Y 481.717,Z 361.477,A -85,B 0,C 180,E1 -6768.721,E2 -6768.721} C_VEL
LIN {X 0,Y 481.651,Z 361.491,A -85,B 0,C 180,E1 -6771.394,E2 -6771.394} C_VEL
LIN {X 0,Y 481.681,Z 361.48,A -85,B 0,C 180,E1 -6774.112,E2 -6774.112} C_VEL
LIN {X 0,Y 481.749,Z 361.479,A -85,B 0,C 180,E1 -6777.138,E2 -6777.138} C_VEL
LIN {X 0,Y 481.681,Z 361.482,A -85,B 0,C 180,E1 -6779.74,E2 -6779.74} C_VEL
LIN {X 0,Y 481.675,Z 361.483,A -85,B 0,C 180,E1 -6782.673,E2 -6782.673} C_VEL
LIN {X 0,Y 481.644,Z 361.486,A -85,B 0,C 180,E1 -6785.708,E2 -6785.708} C_VEL
LIN {X 0,Y 481.691,Z 361.484,A -85,B 0,C 180,E1 -6788.856,E2 -6788.856} C_VEL
LIN {X 0,Y 481.646,Z 361.484,A -85,B 0,C 180,E1 -6792.16,E2 -6792.16} C_VEL
LIN {X 0,Y 481.658,Z 361.485,A -85,B 0,C 180,E1 -6795.542,E2 -6795.542} C_VEL
LIN {X 0,Y 481.66,Z 361.483,A -85,B 0,C 180,E1 -6798.085,E2 -6798.085} C_VEL
LIN {X 0,Y 481.688,Z 361.485,A -85,B 0,C 180,E1 -6801.142,E2 -6801.142} C_VEL
LIN {X 0,Y 481.663,Z 361.489,A -85,B 0,C 180,E1 -6804.794,E2 -6804.794} C_VEL
LIN {X 0,Y 481.668,Z 361.484,A -85,B 0,C 180,E1 -6807.325,E2 -6807.325} C_VEL
LIN {X 0,Y 481.673,Z 361.482,A -85,B 0,C 180,E1 -6810.258,E2 -6810.258} C_VEL
LIN {X 0,Y 481.746,Z 361.476,A -85,B 0,C 180,E1 -6813.112,E2 -6813.112} C_VEL
LIN {X 0,Y 481.67,Z 361.481,A -85,B 0,C 180,E1 -6815.886,E2 -6815.886} C_VEL
LIN {X 0,Y 481.695,Z 361.483,A -85,B 0,C 180,E1 -6819.027,E2 -6819.027} C_VEL
LIN {X 0,Y 481.7,Z 361.479,A -85,B 0,C 180,E1 -6822.158,E2 -6822.158} C_VEL
LIN {X 0,Y 481.734,Z 361.481,A -85,B 0,C 180,E1 -6824.775,E2 -6824.775} C_VEL
LIN {X 0,Y 481.744,Z 361.475,A -85,B 0,C 180,E1 -6828.215,E2 -6828.215} C_VEL
LIN {X 0,Y 481.755,Z 361.471,A -85,B 0,C 180,E1 -6831.611,E2 -6831.611} C_VEL
LIN {X 0,Y 481.813,Z 361.466,A -85,B 0,C 180,E1 -6834.139,E2 -6834.139} C_VEL
LIN {X 0,Y 481.92,Z 361.45,A -85,B 0,C 180,E1 -6837.492,E2 -6837.492} C_VEL
LIN {X 0,Y 481.917,Z 361.455,A -85,B 0,C 180,E1 -6840.835,E2 -6840.835} C_VEL
LIN {X 0,Y 481.92,Z 361.459,A -85,B 0,C 180,E1 -6842.507,E2 -6842.507} C_VEL
LIN {X 0,Y 481.807,Z 361.465,A -85,B 0,C 180,E1 -6845.86,E2 -6845.86} C_VEL
LIN {X 0,Y 481.755,Z 361.479,A -85,B 0,C 180,E1 -6848.388,E2 -6848.388} C_VEL
LIN {X 0,Y 481.743,Z 361.473,A -85,B 0,C 180,E1 -6851.785,E2 -6851.785} C_VEL
LIN {X 0,Y 481.733,Z 361.473,A -85,B 0,C 180,E1 -6855.224,E2 -6855.224} C_VEL
LIN {X 0,Y 481.703,Z 361.48,A -85,B 0,C 180,E1 -6858.722,E2 -6858.722} C_VEL
LIN {X 0,Y 481.638,Z 361.485,A -85,B 0,C 180,E1 -6861.395,E2 -6861.395} C_VEL
LIN {X 0,Y 481.669,Z 361.488,A -85,B 0,C 180,E1 -6864.113,E2 -6864.113} C_VEL
LIN {X 0,Y 481.744,Z 361.472,A -85,B 0,C 180,E1 -6867.141,E2 -6867.141} C_VEL
LIN {X 0,Y 481.681,Z 361.482,A -85,B 0,C 180,E1 -6869.741,E2 -6869.741} C_VEL
LIN {X 0,Y 481.667,Z 361.484,A -85,B 0,C 180,E1 -6872.675,E2 -6872.675} C_VEL
LIN {X 0,Y 481.637,Z 361.488,A -85,B 0,C 180,E1 -6875.71,E2 -6875.71} C_VEL
LIN {X 0,Y 481.714,Z 361.476,A -85,B 0,C 180,E1 -6879.355,E2 -6879.355} C_VEL
LIN {X 0,Y 481.668,Z 361.489,A -85,B 0,C 180,E1 -6882.159,E2 -6882.159} C_VEL
LIN {X 0,Y 481.655,Z 361.486,A -85,B 0,C 180,E1 -6884.458,E2 -6884.458} C_VEL
LIN {X 0,Y 481.645,Z 361.491,A -85,B 0,C 180,E1 -6887.84,E2 -6887.84} C_VEL
LIN {X 0,Y 481.72,Z 361.476,A -85,B 0,C 180,E1 -6890.646,E2 -6890.646} C_VEL
LIN {X 0,Y 481.641,Z 361.488,A -85,B 0,C 180,E1 -6894.292,E2 -6894.292} C_VEL
LIN {X 0,Y 481.672,Z 361.483,A -85,B 0,C 180,E1 -6897.327,E2 -6897.327} C_VEL
LIN {X 0,Y 481.688,Z 361.487,A -85,B 0,C 180,E1 -6900.26,E2 -6900.26} C_VEL
LIN {X 0,Y 481.726,Z 361.483,A -85,B 0,C 180,E1 -6903.579,E2 -6903.579} C_VEL
LIN {X 0,Y 481.753,Z 361.565,A -85,B 0,C 180,E1 -6903.814,E2 -6903.814} C_VEL
LIN {X 0,Y 483.887,Z 372.524,A -85,B 0,C 180,E1 -6905.777,E2 -6905.777} C_VEL
LIN {X 0,Y 483.606,Z 383.306,A -85,B 0,C 180,E1 -6907.575,E2 -6907.575} C_VEL
LIN {X 0,Y 482.807,Z 403.294,A -85,B 0,C 180,E1 -6910.855,E2 -6910.855} C_VEL
LIN {X 0,Y 482.285,Z 419.656,A -85,B 0,C 180,E1 -6913.497,E2 -6913.497} C_VEL
LIN {X 0,Y 484.83,Z 437.415,A -85,B 0,C 180,E1 -6913.85,E2 -6913.85} C_VEL
LIN {X 0,Y 484.208,Z 528.586,A -85,B 0,C 180,E1 -6915.232,E2 -6915.232} C_VEL
LIN {X 0,Y 483.859,Z 541.719,A -85,B 0,C 180,E1 -6915.597,E2 -6915.597} C_VEL
LIN {X 0,Y 483.438,Z 554.39,A -85,B 0,C 180,E1 -6916.122,E2 -6916.122} C_VEL
LIN {X 0,Y 483.052,Z 565.666,A -85,B 0,C 180,E1 -6916.754,E2 -6916.754} C_VEL
LIN {X 0,Y 482.56,Z 577.432,A -85,B 0,C 180,E1 -6917.603,E2 -6917.603} C_VEL
LIN {X 0,Y 482.184,Z 587.845,A -85,B 0,C 180,E1 -6918.546,E2 -6918.546} C_VEL
LIN {X 0,Y 481.82,Z 596.437,A -85,B 0,C 180,E1 -6919.495,E2 -6919.495} C_VEL
LIN {X 0,Y 481.462,Z 604.363,A -85,B 0,C 180,E1 -6920.548,E2 -6920.548} C_VEL
LIN {X 0,Y 481.203,Z 612.11,A -85,B 0,C 180,E1 -6921.813,E2 -6921.813} C_VEL
LIN {X 0,Y 481.019,Z 619.246,A -85,B 0,C 180,E1 -6923.288,E2 -6923.288} C_VEL
LIN {X 0,Y 480.932,Z 623.994,A -85,B 0,C 180,E1 -6924.55,E2 -6924.55} C_VEL
LIN {X 0,Y 480.844,Z 627.618,A -85,B 0,C 180,E1 -6925.809,E2 -6925.809} C_VEL
LIN {X 0,Y 480.893,Z 629.492,A -85,B 0,C 180,E1 -6926.649,E2 -6926.649} C_VEL
LIN {X 0,Y 480.845,Z 630.892,A -85,B 0,C 180,E1 -6927.487,E2 -6927.487} C_VEL
LIN {X 0,Y 480.823,Z 631.89,A -85,B 0,C 180,E1 -6928.325,E2 -6928.325} C_VEL
LIN {X 0,Y 480.745,Z 632.709,A -85,B 0,C 180,E1 -6930,E2 -6930} C_VEL
LIN {X 0,Y 480.823,Z 631.877,A -85,B 0,C 180,E1 -6931.675,E2 -6931.675} C_VEL
LIN {X 0,Y 480.845,Z 630.873,A -85,B 0,C 180,E1 -6932.513,E2 -6932.513} C_VEL
LIN {X 0,Y 480.893,Z 629.466,A -85,B 0,C 180,E1 -6933.351,E2 -6933.351} C_VEL
LIN {X 0,Y 480.84,Z 626.503,A -85,B 0,C 180,E1 -6934.611,E2 -6934.611} C_VEL
LIN {X 0,Y 480.928,Z 622.504,A -85,B 0,C 180,E1 -6935.871,E2 -6935.871} C_VEL
LIN {X 0,Y 481.106,Z 616.357,A -85,B 0,C 180,E1 -6937.343,E2 -6937.343} C_VEL
LIN {X 0,Y 481.3,Z 609.644,A -85,B 0,C 180,E1 -6938.608,E2 -6938.608} C_VEL
LIN {X 0,Y 481.573,Z 601.319,A -85,B 0,C 180,E1 -6939.874,E2 -6939.874} C_VEL
LIN {X 0,Y 481.979,Z 592.796,A -85,B 0,C 180,E1 -6940.927,E2 -6940.927} C_VEL
LIN {X 0,Y 482.436,Z 582.335,A -85,B 0,C 180,E1 -6941.975,E2 -6941.975} C_VEL
LIN {X 0,Y 482.813,Z 570.574,A -85,B 0,C 180,E1 -6942.921,E2 -6942.921} C_VEL
LIN {X 0,Y 483.296,Z 558.527,A -85,B 0,C 180,E1 -6943.668,E2 -6943.668} C_VEL
LIN {X 0,Y 483.733,Z 546.16,A -85,B 0,C 180,E1 -6944.245,E2 -6944.245} C_VEL
LIN {X 0,Y 484.11,Z 533.479,A -85,B 0,C 180,E1 -6944.663,E2 -6944.663} C_VEL
LIN {X 0,Y 484.311,Z 520.248,A -85,B 0,C 180,E1 -6944.926,E2 -6944.926} C_VEL
LIN {X 0,Y 484.811,Z 436.4,A -85,B 0,C 180,E1 -6946.181,E2 -6946.181} C_VEL
LIN {X 0,Y 482.273,Z 419.333,A -85,B 0,C 180,E1 -6946.537,E2 -6946.537} C_VEL
LIN {X 0,Y 483.005,Z 399.514,A -85,B 0,C 180,E1 -6949.773,E2 -6949.773} C_VEL
LIN {X 0,Y 483.727,Z 380.897,A -85,B 0,C 180,E1 -6952.87,E2 -6952.87} C_VEL
LIN {X 0,Y 483.99,Z 372.922,A -85,B 0,C 180,E1 -6954.218,E2 -6954.218} C_VEL
LIN {X 0,Y 481.744,Z 361.48,A -85,B 0,C 180,E1 -6956.361,E2 -6956.361} C_VEL
LIN {X 0,Y 481.688,Z 361.485,A -85,B 0,C 180,E1 -6959.74,E2 -6959.74} C_VEL
LIN {X 0,Y 481.672,Z 361.483,A -85,B 0,C 180,E1 -6962.673,E2 -6962.673} C_VEL
LIN {X 0,Y 481.641,Z 361.49,A -85,B 0,C 180,E1 -6965.708,E2 -6965.708} C_VEL
LIN {X 0,Y 481.72,Z 361.476,A -85,B 0,C 180,E1 -6969.354,E2 -6969.354} C_VEL
LIN {X 0,Y 481.645,Z 361.486,A -85,B 0,C 180,E1 -6972.16,E2 -6972.16} C_VEL
LIN {X 0,Y 481.655,Z 361.487,A -85,B 0,C 180,E1 -6975.542,E2 -6975.542} C_VEL
LIN {X 0,Y 481.669,Z 361.488,A -85,B 0,C 180,E1 -6978.084,E2 -6978.084} C_VEL
LIN {X 0,Y 481.697,Z 361.479,A -85,B 0,C 180,E1 -6981.143,E2 -6981.143} C_VEL
LIN {X 0,Y 481.662,Z 361.483,A -85,B 0,C 180,E1 -6984.794,E2 -6984.794} C_VEL
LIN {X 0,Y 481.667,Z 361.483,A -85,B 0,C 180,E1 -6987.325,E2 -6987.325} C_VEL
LIN {X 0,Y 481.681,Z 361.481,A -85,B 0,C 180,E1 -6990.259,E2 -6990.259} C_VEL
LIN {X 0,Y 481.744,Z 361.473,A -85,B 0,C 180,E1 -6993.112,E2 -6993.112} C_VEL
LIN {X 0,Y 481.669,Z 361.487,A -85,B 0,C 180,E1 -6995.887,E2 -6995.887} C_VEL
LIN {X 0,Y 481.694,Z 361.477,A -85,B 0,C 180,E1 -6999.027,E2 -6999.027} C_VEL
LIN {X 0,Y 481.698,Z 361.476,A -85,B 0,C 180,E1 -7002.158,E2 -7002.158} C_VEL
LIN {X 0,Y 481.735,Z 361.474,A -85,B 0,C 180,E1 -7004.776,E2 -7004.776} C_VEL
LIN {X 0,Y 481.743,Z 361.471,A -85,B 0,C 180,E1 -7008.215,E2 -7008.215} C_VEL
LIN {X 0,Y 481.755,Z 361.472,A -85,B 0,C 180,E1 -7011.612,E2 -7011.612} C_VEL
LIN {X 0,Y 481.808,Z 361.465,A -85,B 0,C 180,E1 -7014.14,E2 -7014.14} C_VEL
LIN {X 0,Y 481.92,Z 361.453,A -85,B 0,C 180,E1 -7017.493,E2 -7017.493} C_VEL
LIN {X 0,Y 481.931,Z 361.451,A -85,B 0,C 180,E1 -7020,E2 -7020} C_VEL
LIN {X 0,Y 481.921,Z 361.447,A -85,B 0,C 180,E1 -7022.508,E2 -7022.508} C_VEL
LIN {X 0,Y 481.814,Z 361.464,A -85,B 0,C 180,E1 -7025.861,E2 -7025.861} C_VEL
LIN {X 0,Y 481.755,Z 361.469,A -85,B 0,C 180,E1 -7028.389,E2 -7028.389} C_VEL
LIN {X 0,Y 481.744,Z 361.47,A -85,B 0,C 180,E1 -7031.785,E2 -7031.785} C_VEL
LIN {X 0,Y 481.734,Z 361.478,A -85,B 0,C 180,E1 -7035.225,E2 -7035.225} C_VEL
LIN {X 0,Y 481.705,Z 361.481,A -85,B 0,C 180,E1 -7038.722,E2 -7038.722} C_VEL
LIN {X 0,Y 481.665,Z 361.487,A -85,B 0,C 180,E1 -7041.394,E2 -7041.394} C_VEL
LIN {X 0,Y 481.675,Z 361.478,A -85,B 0,C 180,E1 -7044.114,E2 -7044.114} C_VEL
LIN {X 0,Y 481.746,Z 361.477,A -85,B 0,C 180,E1 -7047.141,E2 -7047.141} C_VEL
LIN {X 0,Y 481.673,Z 361.481,A -85,B 0,C 180,E1 -7049.742,E2 -7049.742} C_VEL
LIN {X 0,Y 481.668,Z 361.489,A -85,B 0,C 180,E1 -7052.675,E2 -7052.675} C_VEL
LIN {X 0,Y 481.639,Z 361.486,A -85,B 0,C 180,E1 -7055.71,E2 -7055.71} C_VEL
LIN {X 0,Y 481.707,Z 361.479,A -85,B 0,C 180,E1 -7059.354,E2 -7059.354} C_VEL
LIN {X 0,Y 481.672,Z 361.482,A -85,B 0,C 180,E1 -7062.159,E2 -7062.159} C_VEL
LIN {X 0,Y 481.658,Z 361.49,A -85,B 0,C 180,E1 -7064.458,E2 -7064.458} C_VEL
LIN {X 0,Y 481.653,Z 361.485,A -85,B 0,C 180,E1 -7067.841,E2 -7067.841} C_VEL
LIN {X 0,Y 481.68,Z 361.488,A -85,B 0,C 180,E1 -7070.652,E2 -7070.652} C_VEL
LIN {X 0,Y 481.692,Z 361.537,A -85,B 0,C 180,E1 -7073.845,E2 -7073.845} C_VEL
LIN {X 0,Y 482.777,Z 368.226,A -85,B 0,C 180,E1 -7075.408,E2 -7075.408} C_VEL
LIN {X 0,Y 482.466,Z 377.819,A -85,B 0,C 180,E1 -7077.523,E2 -7077.523} C_VEL
LIN {X 0,Y 484.98,Z 389.987,A -85,B 0,C 180,E1 -7077.822,E2 -7077.822} C_VEL
LIN {X 0,Y 484.589,Z 459.892,A -85,B 0,C 180,E1 -7078.873,E2 -7078.873} C_VEL
LIN {X 0,Y 483.843,Z 463.814,A -85,B 0,C 180,E1 -7078.906,E2 -7078.906} C_VEL
LIN {X 0,Y 478.199,Z 476.097,A -85,B 0,C 180,E1 -7078.896,E2 -7078.896} C_VEL
LIN {X 0,Y 477.589,Z 479.999,A -85,B 0,C 180,E1 -7078.943,E2 -7078.943} C_VEL
LIN {X 0,Y 477.389,Z 493.503,A -85,B 0,C 180,E1 -7079.262,E2 -7079.262} C_VEL
LIN {X 0,Y 477.097,Z 505.352,A -85,B 0,C 180,E1 -7079.701,E2 -7079.701} C_VEL
LIN {X 0,Y 476.675,Z 517.98,A -85,B 0,C 180,E1 -7080.354,E2 -7080.354} C_VEL
LIN {X 0,Y 476.256,Z 529.004,A -85,B 0,C 180,E1 -7081.101,E2 -7081.101} C_VEL
LIN {X 0,Y 475.792,Z 539.487,A -85,B 0,C 180,E1 -7081.989,E2 -7081.989} C_VEL
LIN {X 0,Y 475.35,Z 548.779,A -85,B 0,C 180,E1 -7082.959,E2 -7082.959} C_VEL
LIN {X 0,Y 474.918,Z 557.774,A -85,B 0,C 180,E1 -7084.117,E2 -7084.117} C_VEL
LIN {X 0,Y 474.5,Z 566.409,A -85,B 0,C 180,E1 -7085.499,E2 -7085.499} C_VEL
LIN {X 0,Y 474.261,Z 572.637,A -85,B 0,C 180,E1 -7086.748,E2 -7086.748} C_VEL
LIN {X 0,Y 474.017,Z 578.45,A -85,B 0,C 180,E1 -7088.244,E2 -7088.244} C_VEL
LIN {X 0,Y 473.903,Z 582.423,A -85,B 0,C 180,E1 -7089.605,E2 -7089.605} C_VEL
LIN {X 0,Y 473.764,Z 585.241,A -85,B 0,C 180,E1 -7090.953,E2 -7090.953} C_VEL
LIN {X 0,Y 473.719,Z 586.541,A -85,B 0,C 180,E1 -7091.848,E2 -7091.848} C_VEL
LIN {X 0,Y 473.663,Z 587.392,A -85,B 0,C 180,E1 -7092.738,E2 -7092.738} C_VEL
LIN {X 0,Y 473.619,Z 587.781,A -85,B 0,C 180,E1 -7093.624,E2 -7093.624} C_VEL
LIN {X 0,Y 473.668,Z 587.73,A -85,B 0,C 180,E1 -7094.675,E2 -7094.675} C_VEL
LIN {X 0,Y 473.694,Z 586.463,A -85,B 0,C 180,E1 -7096.268,E2 -7096.268} C_VEL
LIN {X 0,Y 473.742,Z 585.17,A -85,B 0,C 180,E1 -7097.143,E2 -7097.143} C_VEL
LIN {X 0,Y 473.867,Z 583.044,A -85,B 0,C 180,E1 -7098.2,E2 -7098.2} C_VEL
LIN {X 0,Y 473.996,Z 578.649,A -85,B 0,C 180,E1 -7099.751,E2 -7099.751} C_VEL
LIN {X 0,Y 474.175,Z 573.747,A -85,B 0,C 180,E1 -7101.047,E2 -7101.047} C_VEL
LIN {X 0,Y 474.467,Z 567.572,A -85,B 0,C 180,E1 -7102.339,E2 -7102.339} C_VEL
LIN {X 0,Y 474.771,Z 559.913,A -85,B 0,C 180,E1 -7103.626,E2 -7103.626} C_VEL
LIN {X 0,Y 475.209,Z 550.298,A -85,B 0,C 180,E1 -7104.909,E2 -7104.909} C_VEL
LIN {X 0,Y 475.694,Z 540.374,A -85,B 0,C 180,E1 -7105.976,E2 -7105.976} C_VEL
LIN {X 0,Y 476.101,Z 529.204,A -85,B 0,C 180,E1 -7106.933,E2 -7106.933} C_VEL
LIN {X 0,Y 476.575,Z 518.228,A -85,B 0,C 180,E1 -7107.676,E2 -7107.676} C_VEL
LIN {X 0,Y 476.954,Z 506.117,A -85,B 0,C 180,E1 -7108.311,E2 -7108.311} C_VEL
LIN {X 0,Y 477.309,Z 493.346,A -85,B 0,C 180,E1 -7108.787,E2 -7108.787} C_VEL
LIN {X 0,Y 477.479,Z 481.421,A -85,B 0,C 180,E1 -7109.078,E2 -7109.078} C_VEL
LIN {X 0,Y 478.121,Z 391.095,A -85,B 0,C 180,E1 -7110.453,E2 -7110.453} C_VEL
LIN {X 0,Y 475.416,Z 377.989,A -85,B 0,C 180,E1 -7110.752,E2 -7110.752} C_VEL
LIN {X 0,Y 475.754,Z 367.945,A -85,B 0,C 180,E1 -7112.964,E2 -7112.964} C_VEL
LIN {X 0,Y 474.653,Z 362.361,A -85,B 0,C 180,E1 -7114.299,E2 -7114.299} C_VEL
LIN {X 0,Y 474.71,Z 362.353,A -85,B 0,C 180,E1 -7116.802,E2 -7116.802} C_VEL
LIN {X 0,Y 474.709,Z 362.357,A -85,B 0,C 180,E1 -7119.372,E2 -7119.372} C_VEL
LIN {X 0,Y 474.707,Z 362.349,A -85,B 0,C 180,E1 -7122.276,E2 -7122.276} C_VEL
LIN {X 0,Y 474.686,Z 362.354,A -85,B 0,C 180,E1 -7125.767,E2 -7125.767} C_VEL
LIN {X 0,Y 474.669,Z 362.358,A -85,B 0,C 180,E1 -7129.01,E2 -7129.01} C_VEL
LIN {X 0,Y 474.595,Z 362.365,A -85,B 0,C 180,E1 -7131.728,E2 -7131.728} C_VEL
LIN {X 0,Y 474.663,Z 362.355,A -85,B 0,C 180,E1 -7134.492,E2 -7134.492} C_VEL
LIN {X 0,Y 474.683,Z 362.358,A -85,B 0,C 180,E1 -7137.334,E2 -7137.334} C_VEL
LIN {X 0,Y 474.614,Z 362.364,A -85,B 0,C 180,E1 -7140.811,E2 -7140.811} C_VEL
LIN {X 0,Y 474.639,Z 362.357,A -85,B 0,C 180,E1 -7143.983,E2 -7143.983} C_VEL
LIN {X 0,Y 474.576,Z 362.37,A -85,B 0,C 180,E1 -7146.899,E2 -7146.899} C_VEL
LIN {X 0,Y 474.627,Z 362.36,A -85,B 0,C 180,E1 -7149.647,E2 -7149.647} C_VEL
LIN {X 0,Y 474.63,Z 362.365,A -85,B 0,C 180,E1 -7152.931,E2 -7152.931} C_VEL
LIN {X 0,Y 474.615,Z 362.36,A -85,B 0,C 180,E1 -7155.895,E2 -7155.895} C_VEL
LIN {X 0,Y 474.629,Z 362.366,A -85,B 0,C 180,E1 -7159.039,E2 -7159.039} C_VEL
LIN {X 0,Y 474.611,Z 362.361,A -85,B 0,C 180,E1 -7161.702,E2 -7161.702} C_VEL
LIN {X 0,Y 474.625,Z 362.365,A -85,B 0,C 180,E1 -7164.725,E2 -7164.725} C_VEL
LIN {X 0,Y 474.632,Z 362.358,A -85,B 0,C 180,E1 -7167.787,E2 -7167.787} C_VEL
LIN {X 0,Y 474.619,Z 362.368,A -85,B 0,C 180,E1 -7170.884,E2 -7170.884} C_VEL
LIN {X 0,Y 474.66,Z 362.355,A -85,B 0,C 180,E1 -7173.628,E2 -7173.628} C_VEL
LIN {X 0,Y 474.629,Z 362.365,A -85,B 0,C 180,E1 -7176.64,E2 -7176.64} C_VEL
LIN {X 0,Y 474.649,Z 362.357,A -85,B 0,C 180,E1 -7180.089,E2 -7180.089} C_VEL
LIN {X 0,Y 474.644,Z 362.364,A -85,B 0,C 180,E1 -7182.774,E2 -7182.774} C_VEL
LIN {X 0,Y 474.641,Z 362.357,A -85,B 0,C 180,E1 -7185.42,E2 -7185.42} C_VEL
LIN {X 0,Y 474.697,Z 362.351,A -85,B 0,C 180,E1 -7188.037,E2 -7188.037} C_VEL
LIN {X 0,Y 474.72,Z 362.347,A -85,B 0,C 180,E1 -7191.486,E2 -7191.486} C_VEL
LIN {X 0,Y 474.774,Z 362.342,A -85,B 0,C 180,E1 -7194.052,E2 -7194.052} C_VEL
LIN {X 0,Y 474.886,Z 362.326,A -85,B 0,C 180,E1 -7197.455,E2 -7197.455} C_VEL
LIN {X 0,Y 474.868,Z 362.332,A -85,B 0,C 180,E1 -7200.848,E2 -7200.848} C_VEL
LIN {X 0,Y 474.886,Z 362.334,A -85,B 0,C 180,E1 -7202.544,E2 -7202.544} C_VEL
LIN {X 0,Y 474.77,Z 362.343,A -85,B 0,C 180,E1 -7205.948,E2 -7205.948} C_VEL
LIN {X 0,Y 474.72,Z 362.354,A -85,B 0,C 180,E1 -7208.514,E2 -7208.514} C_VEL
LIN {X 0,Y 474.696,Z 362.353,A -85,B 0,C 180,E1 -7211.962,E2 -7211.962} C_VEL
LIN {X 0,Y 474.692,Z 362.352,A -85,B 0,C 180,E1 -7215.777,E2 -7215.777} C_VEL
LIN {X 0,Y 474.657,Z 362.356,A -85,B 0,C 180,E1 -7219.01,E2 -7219.01} C_VEL
LIN {X 0,Y 474.582,Z 362.366,A -85,B 0,C 180,E1 -7221.729,E2 -7221.729} C_VEL
LIN {X 0,Y 474.651,Z 362.361,A -85,B 0,C 180,E1 -7224.493,E2 -7224.493} C_VEL
LIN {X 0,Y 474.691,Z 362.351,A -85,B 0,C 180,E1 -7227.339,E2 -7227.339} C_VEL
LIN {X 0,Y 474.603,Z 362.363,A -85,B 0,C 180,E1 -7230.812,E2 -7230.812} C_VEL
LIN {X 0,Y 474.632,Z 362.364,A -85,B 0,C 180,E1 -7233.985,E2 -7233.985} C_VEL
LIN {X 0,Y 474.57,Z 362.366,A -85,B 0,C 180,E1 -7236.901,E2 -7236.901} C_VEL
LIN {X 0,Y 474.649,Z 362.359,A -85,B 0,C 180,E1 -7239.652,E2 -7239.652} C_VEL
LIN {X 0,Y 474.646,Z 362.356,A -85,B 0,C 180,E1 -7242.931,E2 -7242.931} C_VEL
LIN {X 0,Y 474.605,Z 362.368,A -85,B 0,C 180,E1 -7245.896,E2 -7245.896} C_VEL
LIN {X 0,Y 474.638,Z 362.357,A -85,B 0,C 180,E1 -7249.039,E2 -7249.039} C_VEL
LIN {X 0,Y 474.617,Z 362.365,A -85,B 0,C 180,E1 -7251.703,E2 -7251.703} C_VEL
LIN {X 0,Y 474.628,Z 362.359,A -85,B 0,C 180,E1 -7254.727,E2 -7254.727} C_VEL
LIN {X 0,Y 474.637,Z 362.365,A -85,B 0,C 180,E1 -7257.789,E2 -7257.789} C_VEL
LIN {X 0,Y 474.632,Z 362.363,A -85,B 0,C 180,E1 -7260.883,E2 -7260.883} C_VEL
LIN {X 0,Y 474.725,Z 362.507,A -85,B 0,C 180,E1 -7263.633,E2 -7263.633} C_VEL
LIN {X 0,Y 477.028,Z 374.849,A -85,B 0,C 180,E1 -7265.873,E2 -7265.873} C_VEL
LIN {X 0,Y 476.323,Z 390.988,A -85,B 0,C 180,E1 -7268.582,E2 -7268.582} C_VEL
LIN {X 0,Y 475.627,Z 409.782,A -85,B 0,C 180,E1 -7271.7,E2 -7271.7} C_VEL
LIN {X 0,Y 475.306,Z 419.378,A -85,B 0,C 180,E1 -7273.259,E2 -7273.259} C_VEL
LIN {X 0,Y 477.988,Z 437.912,A -85,B 0,C 180,E1 -7273.634,E2 -7273.634} C_VEL
LIN {X 0,Y 477.331,Z 527.979,A -85,B 0,C 180,E1 -7275.014,E2 -7275.014} C_VEL
LIN {X 0,Y 476.974,Z 541.219,A -85,B 0,C 180,E1 -7275.385,E2 -7275.385} C_VEL
LIN {X 0,Y 476.541,Z 553.944,A -85,B 0,C 180,E1 -7275.917,E2 -7275.917} C_VEL
LIN {X 0,Y 476.102,Z 565.249,A -85,B 0,C 180,E1 -7276.556,E2 -7276.556} C_VEL
LIN {X 0,Y 475.603,Z 576.704,A -85,B 0,C 180,E1 -7277.392,E2 -7277.392} C_VEL
LIN {X 0,Y 475.198,Z 587.459,A -85,B 0,C 180,E1 -7278.375,E2 -7278.375} C_VEL
LIN {X 0,Y 474.779,Z 596.059,A -85,B 0,C 180,E1 -7279.337,E2 -7279.337} C_VEL
LIN {X 0,Y 474.434,Z 603.995,A -85,B 0,C 180,E1 -7280.407,E2 -7280.407} C_VEL
LIN {X 0,Y 474.151,Z 611.751,A -85,B 0,C 180,E1 -7281.691,E2 -7281.691} C_VEL
LIN {X 0,Y 473.934,Z 618.892,A -85,B 0,C 180,E1 -7283.187,E2 -7283.187} C_VEL
LIN {X 0,Y 473.846,Z 623.646,A -85,B 0,C 180,E1 -7284.468,E2 -7284.468} C_VEL
LIN {X 0,Y 473.748,Z 627.275,A -85,B 0,C 180,E1 -7285.746,E2 -7285.746} C_VEL
LIN {X 0,Y 473.801,Z 629.152,A -85,B 0,C 180,E1 -7286.599,E2 -7286.599} C_VEL
LIN {X 0,Y 473.761,Z 630.555,A -85,B 0,C 180,E1 -7287.449,E2 -7287.449} C_VEL
LIN {X 0,Y 473.756,Z 631.555,A -85,B 0,C 180,E1 -7288.3,E2 -7288.3} C_VEL
LIN {X 0,Y 473.672,Z 632.377,A -85,B 0,C 180,E1 -7290,E2 -7290} C_VEL
LIN {X 0,Y 473.756,Z 631.547,A -85,B 0,C 180,E1 -7291.7,E2 -7291.7} C_VEL
LIN {X 0,Y 473.761,Z 630.542,A -85,B 0,C 180,E1 -7292.551,E2 -7292.551} C_VEL
LIN {X 0,Y 473.801,Z 629.136,A -85,B 0,C 180,E1 -7293.401,E2 -7293.401} C_VEL
LIN {X 0,Y 473.763,Z 626.176,A -85,B 0,C 180,E1 -7294.68,E2 -7294.68} C_VEL
LIN {X 0,Y 473.834,Z 622.177,A -85,B 0,C 180,E1 -7295.959,E2 -7295.959} C_VEL
LIN {X 0,Y 474.015,Z 616.033,A -85,B 0,C 180,E1 -7297.454,E2 -7297.454} C_VEL
LIN {X 0,Y 474.227,Z 609.322,A -85,B 0,C 180,E1 -7298.737,E2 -7298.737} C_VEL
LIN {X 0,Y 474.541,Z 601.001,A -85,B 0,C 180,E1 -7300.021,E2 -7300.021} C_VEL
LIN {X 0,Y 474.974,Z 592.482,A -85,B 0,C 180,E1 -7301.09,E2 -7301.09} C_VEL
LIN {X 0,Y 475.436,Z 582.253,A -85,B 0,C 180,E1 -7302.133,E2 -7302.133} C_VEL
LIN {X 0,Y 475.806,Z 571.872,A -85,B 0,C 180,E1 -7302.996,E2 -7302.996} C_VEL
LIN {X 0,Y 476.332,Z 560.222,A -85,B 0,C 180,E1 -7303.763,E2 -7303.763} C_VEL
LIN {X 0,Y 476.797,Z 548.606,A -85,B 0,C 180,E1 -7304.348,E2 -7304.348} C_VEL
LIN {X 0,Y 477.205,Z 535.259,A -85,B 0,C 180,E1 -7304.826,E2 -7304.826} C_VEL
LIN {X 0,Y 477.48,Z 522.218,A -85,B 0,C 180,E1 -7305.117,E2 -7305.117} C_VEL
LIN {X 0,Y 477.992,Z 437.06,A -85,B 0,C 180,E1 -7306.415,E2 -7306.415} C_VEL
LIN {X 0,Y 475.318,Z 418.908,A -85,B 0,C 180,E1 -7306.813,E2 -7306.813} C_VEL
LIN {X 0,Y 476.061,Z 399.295,A -85,B 0,C 180,E1 -7310.074,E2 -7310.074} C_VEL
LIN {X 0,Y 476.873,Z 380.722,A -85,B 0,C 180,E1 -7313.218,E2 -7313.218} C_VEL
LIN {X 0,Y 477.018,Z 374.092,A -85,B 0,C 180,E1 -7314.363,E2 -7314.363} C_VEL
LIN {X 0,Y 474.938,Z 363.494,A -85,B 0,C 180,E1 -7316.354,E2 -7316.354} C_VEL
LIN {X 0,Y 474.689,Z 362.357,A -85,B 0,C 180,E1 -7316.606,E2 -7316.606} C_VEL
LIN {X 0,Y 474.63,Z 362.363,A -85,B 0,C 180,E1 -7319.251,E2 -7319.251} C_VEL
LIN {X 0,Y 474.616,Z 362.365,A -85,B 0,C 180,E1 -7322.43,E2 -7322.43} C_VEL
LIN {X 0,Y 474.618,Z 362.363,A -85,B 0,C 180,E1 -7325.47,E2 -7325.47} C_VEL
LIN {X 0,Y 474.623,Z 362.361,A -85,B 0,C 180,E1 -7328.455,E2 -7328.455} C_VEL
LIN {X 0,Y 474.638,Z 362.359,A -85,B 0,C 180,E1 -7330.961,E2 -7330.961} C_VEL
LIN {X 0,Y 474.605,Z 362.369,A -85,B 0,C 180,E1 -7334.104,E2 -7334.104} C_VEL
LIN {X 0,Y 474.646,Z 362.358,A -85,B 0,C 180,E1 -7337.069,E2 -7337.069} C_VEL
LIN {X 0,Y 474.668,Z 362.355,A -85,B 0,C 180,E1 -7340.456,E2 -7340.456} C_VEL
LIN {X 0,Y 474.587,Z 362.368,A -85,B 0,C 180,E1 -7343.676,E2 -7343.676} C_VEL
LIN {X 0,Y 474.636,Z 362.356,A -85,B 0,C 180,E1 -7346.779,E2 -7346.779} C_VEL
LIN {X 0,Y 474.607,Z 362.365,A -85,B 0,C 180,E1 -7349.77,E2 -7349.77} C_VEL
LIN {X 0,Y 474.707,Z 362.349,A -85,B 0,C 180,E1 -7352.68,E2 -7352.68} C_VEL
LIN {X 0,Y 474.651,Z 362.36,A -85,B 0,C 180,E1 -7355.507,E2 -7355.507} C_VEL
LIN {X 0,Y 474.662,Z 362.354,A -85,B 0,C 180,E1 -7359.185,E2 -7359.185} C_VEL
LIN {X 0,Y 474.648,Z 362.357,A -85,B 0,C 180,E1 -7361.884,E2 -7361.884} C_VEL
LIN {X 0,Y 474.691,Z 362.351,A -85,B 0,C 180,E1 -7364.544,E2 -7364.544} C_VEL
LIN {X 0,Y 474.696,Z 362.35,A -85,B 0,C 180,E1 -7368.038,E2 -7368.038} C_VEL
LIN {X 0,Y 474.72,Z 362.35,A -85,B 0,C 180,E1 -7371.486,E2 -7371.486} C_VEL
LIN {X 0,Y 474.77,Z 362.342,A -85,B 0,C 180,E1 -7374.052,E2 -7374.052} C_VEL
LIN {X 0,Y 474.886,Z 362.329,A -85,B 0,C 180,E1 -7377.456,E2 -7377.456} C_VEL
LIN {X 0,Y 474.869,Z 362.332,A -85,B 0,C 180,E1 -7380.848,E2 -7380.848} C_VEL
LIN {X 0,Y 474.887,Z 362.323,A -85,B 0,C 180,E1 -7382.545,E2 -7382.545} C_VEL
LIN {X 0,Y 474.775,Z 362.34,A -85,B 0,C 180,E1 -7385.948,E2 -7385.948} C_VEL
LIN {X 0,Y 474.721,Z 362.346,A -85,B 0,C 180,E1 -7388.514,E2 -7388.514} C_VEL
LIN {X 0,Y 474.697,Z 362.347,A -85,B 0,C 180,E1 -7391.963,E2 -7391.963} C_VEL
LIN {X 0,Y 474.691,Z 362.352,A -85,B 0,C 180,E1 -7395.456,E2 -7395.456} C_VEL
LIN {X 0,Y 474.658,Z 362.363,A -85,B 0,C 180,E1 -7399.011,E2 -7399.011} C_VEL
LIN {X 0,Y 474.602,Z 362.364,A -85,B 0,C 180,E1 -7401.729,E2 -7401.729} C_VEL
LIN {X 0,Y 474.655,Z 362.355,A -85,B 0,C 180,E1 -7404.493,E2 -7404.493} C_VEL
LIN {X 0,Y 474.693,Z 362.354,A -85,B 0,C 180,E1 -7407.34,E2 -7407.34} C_VEL
LIN {X 0,Y 474.6,Z 362.368,A -85,B 0,C 180,E1 -7410.811,E2 -7410.811} C_VEL
LIN {X 0,Y 474.633,Z 362.353,A -85,B 0,C 180,E1 -7413.985,E2 -7413.985} C_VEL
LIN {X 0,Y 474.571,Z 362.374,A -85,B 0,C 180,E1 -7416.901,E2 -7416.901} C_VEL
LIN {X 0,Y 474.644,Z 362.357,A -85,B 0,C 180,E1 -7419.652,E2 -7419.652} C_VEL
LIN {X 0,Y 474.65,Z 362.362,A -85,B 0,C 180,E1 -7422.931,E2 -7422.931} C_VEL
LIN {X 0,Y 474.613,Z 362.362,A -85,B 0,C 180,E1 -7425.897,E2 -7425.897} C_VEL
LIN {X 0,Y 474.631,Z 362.365,A -85,B 0,C 180,E1 -7429.041,E2 -7429.041} C_VEL
LIN {X 0,Y 474.611,Z 362.368,A -85,B 0,C 180,E1 -7431.705,E2 -7431.705} C_VEL
LIN {X 0,Y 474.643,Z 362.463,A -85,B 0,C 180,E1 -7433.655,E2 -7433.655} C_VEL
LIN {X 0,Y 475.84,Z 369.575,A -85,B 0,C 180,E1 -7435.347,E2 -7435.347} C_VEL
LIN {X 0,Y 475.524,Z 378.328,A -85,B 0,C 180,E1 -7437.281,E2 -7437.281} C_VEL
LIN {X 0,Y 478.236,Z 391.078,A -85,B 0,C 180,E1 -7437.585,E2 -7437.585} C_VEL
LIN {X 0,Y 477.589,Z 479.999,A -85,B 0,C 180,E1 -7438.943,E2 -7438.943} C_VEL
LIN {X 0,Y 477.266,Z 483.882,A -85,B 0,C 180,E1 -7439.003,E2 -7439.003} C_VEL
LIN {X 0,Y 475.937,Z 489.601,A -85,B 0,C 180,E1 -7439.095,E2 -7439.095} C_VEL
LIN {X 0,Y 471.44,Z 502.53,A -85,B 0,C 180,E1 -7439.382,E2 -7439.382} C_VEL
LIN {X 0,Y 470.272,Z 508.11,A -85,B 0,C 180,E1 -7439.591,E2 -7439.591} C_VEL
LIN {X 0,Y 470.126,Z 509.899,A -85,B 0,C 180,E1 -7439.676,E2 -7439.676} C_VEL
LIN {X 0,Y 469.737,Z 520.983,A -85,B 0,C 180,E1 -7440.304,E2 -7440.304} C_VEL
LIN {X 0,Y 469.27,Z 532.186,A -85,B 0,C 180,E1 -7441.12,E2 -7441.12} C_VEL
LIN {X 0,Y 468.736,Z 542.719,A -85,B 0,C 180,E1 -7442.085,E2 -7442.085} C_VEL
LIN {X 0,Y 468.234,Z 552.853,A -85,B 0,C 180,E1 -7443.239,E2 -7443.239} C_VEL
LIN {X 0,Y 467.799,Z 561.303,A -85,B 0,C 180,E1 -7444.435,E2 -7444.435} C_VEL
LIN {X 0,Y 467.396,Z 569.112,A -85,B 0,C 180,E1 -7445.812,E2 -7445.812} C_VEL
LIN {X 0,Y 467.175,Z 574.433,A -85,B 0,C 180,E1 -7446.975,E2 -7446.975} C_VEL
LIN {X 0,Y 466.935,Z 579.487,A -85,B 0,C 180,E1 -7448.361,E2 -7448.361} C_VEL
LIN {X 0,Y 466.788,Z 583.276,A -85,B 0,C 180,E1 -7449.74,E2 -7449.74} C_VEL
LIN {X 0,Y 466.69,Z 585.171,A -85,B 0,C 180,E1 -7450.653,E2 -7450.653} C_VEL
LIN {X 0,Y 466.643,Z 586.602,A -85,B 0,C 180,E1 -7451.593,E2 -7451.593} C_VEL
LIN {X 0,Y 466.587,Z 587.531,A -85,B 0,C 180,E1 -7452.468,E2 -7452.468} C_VEL
LIN {X 0,Y 466.532,Z 588.071,A -85,B 0,C 180,E1 -7453.368,E2 -7453.368} C_VEL
LIN {X 0,Y 466.589,Z 588.082,A -85,B 0,C 180,E1 -7454.581,E2 -7454.581} C_VEL
LIN {X 0,Y 466.595,Z 587.083,A -85,B 0,C 180,E1 -7456.055,E2 -7456.055} C_VEL
